LIN {X 0,Y 450.655,Z 566.335,A -85,B 0,C 180,E1 -8884.109,E2 -8884.109} C_VEL
LIN {X 0,Y 449.557,Z 588.314,A -85,B 0,C 180,E1 -8887.411,E2 -8887.411} C_VEL
LIN {X 0,Y 448.704,Z 611.584,A -85,B 0,C 180,E1 -8890.796,E2 -8890.796} C_VEL
LIN {X 0,Y 448.44,Z 622.118,A -85,B 0,C 180,E1 -8892.238,E2 -8892.238} C_VEL
LIN {X 0,Y 450.986,Z 639.711,A -85,B 0,C 180,E1 -8892.631,E2 -8892.631} C_VEL
LIN {X 0,Y 450.667,Z 684.89,A -85,B 0,C 180,E1 -8893.36,E2 -8893.36} C_VEL
LIN {X 0,Y 449.966,Z 688.81,A -85,B 0,C 180,E1 -8893.398,E2 -8893.398} C_VEL
LIN {X 0,Y 444.273,Z 701.08,A -85,B 0,C 180,E1 -8893.381,E2 -8893.381} C_VEL
LIN {X 0,Y 443.65,Z 704.994,A -85,B 0,C 180,E1 -8893.422,E2 -8893.422} C_VEL
LIN {X 0,Y 443.312,Z 733.868,A -85,B 0,C 180,E1 -8893.922,E2 -8893.922} C_VEL
LIN {X 0,Y 442.949,Z 746.723,A -85,B 0,C 180,E1 -8894.322,E2 -8894.322} C_VEL
LIN {X 0,Y 442.385,Z 759.614,A -85,B 0,C 180,E1 -8894.921,E2 -8894.921} C_VEL
LIN {X 0,Y 441.872,Z 770.653,A -85,B 0,C 180,E1 -8895.61,E2 -8895.61} C_VEL
LIN {X 0,Y 441.394,Z 780.851,A -85,B 0,C 180,E1 -8896.417,E2 -8896.417} C_VEL
LIN {X 0,Y 440.796,Z 791.331,A -85,B 0,C 180,E1 -8897.453,E2 -8897.453} C_VEL
LIN {X 0,Y 440.188,Z 799.921,A -85,B 0,C 180,E1 -8898.487,E2 -8898.487} C_VEL
LIN {X 0,Y 439.608,Z 809.259,A -85,B 0,C 180,E1 -8899.871,E2 -8899.871} C_VEL
LIN {X 0,Y 439.155,Z 816.688,A -85,B 0,C 180,E1 -8901.255,E2 -8901.255} C_VEL
LIN {X 0,Y 438.787,Z 822.657,A -85,B 0,C 180,E1 -8902.638,E2 -8902.638} C_VEL
LIN {X 0,Y 438.678,Z 827.373,A -85,B 0,C 180,E1 -8904.022,E2 -8904.022} C_VEL
LIN {X 0,Y 438.409,Z 830.987,A -85,B 0,C 180,E1 -8905.402,E2 -8905.402} C_VEL
LIN {X 0,Y 438.405,Z 832.844,A -85,B 0,C 180,E1 -8906.323,E2 -8906.323} C_VEL
LIN {X 0,Y 438.391,Z 834.266,A -85,B 0,C 180,E1 -8907.243,E2 -8907.243} C_VEL
LIN {X 0,Y 438.255,Z 835.881,A -85,B 0,C 180,E1 -8909.08,E2 -8909.08} C_VEL
LIN {X 0,Y 438.254,Z 836.117,A -85,B 0,C 180,E1 -8909.999,E2 -8909.999} C_VEL
LIN {X 0,Y 438.255,Z 835.929,A -85,B 0,C 180,E1 -8910.918,E2 -8910.918} C_VEL
LIN {X 0,Y 438.391,Z 834.379,A -85,B 0,C 180,E1 -8912.756,E2 -8912.756} C_VEL
LIN {X 0,Y 438.404,Z 833.019,A -85,B 0,C 180,E1 -8913.676,E2 -8913.676} C_VEL
LIN {X 0,Y 438.474,Z 830.154,A -85,B 0,C 180,E1 -8915.057,E2 -8915.057} C_VEL
LIN {X 0,Y 438.686,Z 825.559,A -85,B 0,C 180,E1 -8916.646,E2 -8916.646} C_VEL
LIN {X 0,Y 438.996,Z 819.257,A -85,B 0,C 180,E1 -8918.283,E2 -8918.283} C_VEL
LIN {X 0,Y 439.4,Z 812.443,A -85,B 0,C 180,E1 -8919.667,E2 -8919.667} C_VEL
LIN {X 0,Y 439.914,Z 803.901,A -85,B 0,C 180,E1 -8921.052,E2 -8921.052} C_VEL
LIN {X 0,Y 440.558,Z 795.158,A -85,B 0,C 180,E1 -8922.202,E2 -8922.202} C_VEL
LIN {X 0,Y 441.142,Z 785.519,A -85,B 0,C 180,E1 -8923.243,E2 -8923.243} C_VEL
LIN {X 0,Y 441.716,Z 774.968,A -85,B 0,C 180,E1 -8924.159,E2 -8924.159} C_VEL
LIN {X 0,Y 442.267,Z 763.215,A -85,B 0,C 180,E1 -8924.964,E2 -8924.964} C_VEL
LIN {X 0,Y 442.817,Z 751.05,A -85,B 0,C 180,E1 -8925.593,E2 -8925.593} C_VEL
LIN {X 0,Y 443.202,Z 738.346,A -85,B 0,C 180,E1 -8926.051,E2 -8926.051} C_VEL
LIN {X 0,Y 443.436,Z 725.465,A -85,B 0,C 180,E1 -8926.338,E2 -8926.338} C_VEL
LIN {X 0,Y 444.112,Z 640.098,A -85,B 0,C 180,E1 -8927.734,E2 -8927.734} C_VEL
LIN {X 0,Y 441.171,Z 622.808,A -85,B 0,C 180,E1 -8928.176,E2 -8928.176} C_VEL
LIN {X 0,Y 441.634,Z 608.028,A -85,B 0,C 180,E1 -8930.492,E2 -8930.492} C_VEL
LIN {X 0,Y 442.46,Z 588.945,A -85,B 0,C 180,E1 -8933.644,E2 -8933.644} C_VEL
LIN {X 0,Y 443.197,Z 571.508,A -85,B 0,C 180,E1 -8936.613,E2 -8936.613} C_VEL
LIN {X 0,Y 443.34,Z 564.171,A -85,B 0,C 180,E1 -8937.88,E2 -8937.88} C_VEL
LIN {X 0,Y 440.924,Z 552.234,A -85,B 0,C 180,E1 -8940.079,E2 -8940.079} C_VEL
LIN {X 0,Y 439.385,Z 545.753,A -85,B 0,C 180,E1 -8941.32,E2 -8941.32} C_VEL
LIN {X 0,Y 439.385,Z 545.755,A -85,B 0,C 180,E1 -8944.042,E2 -8944.042} C_VEL
LIN {X 0,Y 439.354,Z 545.757,A -85,B 0,C 180,E1 -8946.888,E2 -8946.888} C_VEL
LIN {X 0,Y 439.409,Z 545.747,A -85,B 0,C 180,E1 -8949.85,E2 -8949.85} C_VEL
LIN {X 0,Y 439.381,Z 545.75,A -85,B 0,C 180,E1 -8952.626,E2 -8952.626} C_VEL
LIN {X 0,Y 439.397,Z 545.75,A -85,B 0,C 180,E1 -8956.032,E2 -8956.032} C_VEL
LIN {X 0,Y 439.394,Z 545.754,A -85,B 0,C 180,E1 -8959.021,E2 -8959.021} C_VEL
LIN {X 0,Y 439.464,Z 545.804,A -85,B 0,C 180,E1 -8960.616,E2 -8960.616} C_VEL
LIN {X 0,Y 443.64,Z 558.186,A -85,B 0,C 180,E1 -8961.004,E2 -8961.004} C_VEL
LIN {X 0,Y 442.996,Z 626.253,A -85,B 0,C 180,E1 -8962.231,E2 -8962.231} C_VEL
LIN {X 0,Y 442.904,Z 640.237,A -85,B 0,C 180,E1 -8962.685,E2 -8962.685} C_VEL
LIN {X 0,Y 442.685,Z 652.211,A -85,B 0,C 180,E1 -8963.25,E2 -8963.25} C_VEL
LIN {X 0,Y 442.358,Z 664.004,A -85,B 0,C 180,E1 -8963.996,E2 -8963.996} C_VEL
LIN {X 0,Y 441.89,Z 675.616,A -85,B 0,C 180,E1 -8964.932,E2 -8964.932} C_VEL
LIN {X 0,Y 441.419,Z 685.917,A -85,B 0,C 180,E1 -8965.971,E2 -8965.971} C_VEL
LIN {X 0,Y 440.931,Z 695.582,A -85,B 0,C 180,E1 -8967.185,E2 -8967.185} C_VEL
LIN {X 0,Y 440.551,Z 704.101,A -85,B 0,C 180,E1 -8968.503,E2 -8968.503} C_VEL
LIN {X 0,Y 440.109,Z 711.544,A -85,B 0,C 180,E1 -8969.937,E2 -8969.937} C_VEL
LIN {X 0,Y 439.77,Z 717.941,A -85,B 0,C 180,E1 -8971.514,E2 -8971.514} C_VEL
LIN {X 0,Y 439.6,Z 722.254,A -85,B 0,C 180,E1 -8972.894,E2 -8972.894} C_VEL
LIN {X 0,Y 439.415,Z 725.795,A -85,B 0,C 180,E1 -8974.416,E2 -8974.416} C_VEL
LIN {X 0,Y 439.289,Z 727.92,A -85,B 0,C 180,E1 -8975.768,E2 -8975.768} C_VEL
LIN {X 0,Y 439.282,Z 729.321,A -85,B 0,C 180,E1 -8977.42,E2 -8977.42} C_VEL
LIN {X 0,Y 439.291,Z 729.501,A -85,B 0,C 180,E1 -8978.41,E2 -8978.41} C_VEL
LIN {X 0,Y 439.353,Z 729.247,A -85,B 0,C 180,E1 -8979.395,E2 -8979.395} C_VEL
LIN {X 0,Y 439.471,Z 728.221,A -85,B 0,C 180,E1 -8980.647,E2 -8980.647} C_VEL
LIN {X 0,Y 439.647,Z 725.684,A -85,B 0,C 180,E1 -8982.318,E2 -8982.318} C_VEL
LIN {X 0,Y 439.923,Z 722.044,A -85,B 0,C 180,E1 -8983.85,E2 -8983.85} C_VEL
LIN {X 0,Y 440.238,Z 717.703,A -85,B 0,C 180,E1 -8985.201,E2 -8985.201} C_VEL
LIN {X 0,Y 440.71,Z 710.974,A -85,B 0,C 180,E1 -8986.807,E2 -8986.807} C_VEL
LIN {X 0,Y 441.129,Z 704.434,A -85,B 0,C 180,E1 -8988.047,E2 -8988.047} C_VEL
LIN {X 0,Y 441.614,Z 696.861,A -85,B 0,C 180,E1 -8989.223,E2 -8989.223} C_VEL
LIN {X 0,Y 442.106,Z 687.903,A -85,B 0,C 180,E1 -8990.362,E2 -8990.362} C_VEL
LIN {X 0,Y 442.623,Z 677.349,A -85,B 0,C 180,E1 -8991.439,E2 -8991.439} C_VEL
LIN {X 0,Y 443.073,Z 665.968,A -85,B 0,C 180,E1 -8992.366,E2 -8992.366} C_VEL
LIN {X 0,Y 443.499,Z 653.859,A -85,B 0,C 180,E1 -8993.117,E2 -8993.117} C_VEL
LIN {X 0,Y 443.659,Z 640.811,A -85,B 0,C 180,E1 -8993.719,E2 -8993.719} C_VEL
LIN {X 0,Y 443.726,Z 628.913,A -85,B 0,C 180,E1 -8994.091,E2 -8994.091} C_VEL
LIN {X 0,Y 444.376,Z 571.276,A -85,B 0,C 180,E1 -8995.165,E2 -8995.165} C_VEL
LIN {X 0,Y 444.368,Z 558.239,A -85,B 0,C 180,E1 -8995.419,E2 -8995.419} C_VEL
LIN {X 0,Y 439.515,Z 546.251,A -85,B 0,C 180,E1 -8995.902,E2 -8995.902} C_VEL
LIN {X 0,Y 439.442,Z 545.747,A -85,B 0,C 180,E1 -8995.93,E2 -8995.93} C_VEL
LIN {X 0,Y 439.627,Z 545.725,A -85,B 0,C 180,E1 -8998.168,E2 -8998.168} C_VEL
LIN {X 0,Y 439.754,Z 545.709,A -85,B 0,C 180,E1 -9000,E2 -9000} C_VEL
LIN {X 0,Y 439.647,Z 545.724,A -85,B 0,C 180,E1 -9002.749,E2 -9002.749} C_VEL
LIN {X 0,Y 439.612,Z 545.726,A -85,B 0,C 180,E1 -9006.425,E2 -9006.425} C_VEL
LIN {X 0,Y 439.491,Z 545.738,A -85,B 0,C 180,E1 -9009.202,E2 -9009.202} C_VEL
LIN {X 0,Y 439.493,Z 545.738,A -85,B 0,C 180,E1 -9012.727,E2 -9012.727} C_VEL
LIN {X 0,Y 439.436,Z 545.742,A -85,B 0,C 180,E1 -9016.349,E2 -9016.349} C_VEL
LIN {X 0,Y 439.392,Z 545.749,A -85,B 0,C 180,E1 -9019.627,E2 -9019.627} C_VEL
LIN {X 0,Y 439.355,Z 545.76,A -85,B 0,C 180,E1 -9022.576,E2 -9022.576} C_VEL
LIN {X 0,Y 439.395,Z 545.749,A -85,B 0,C 180,E1 -9025.586,E2 -9025.586} C_VEL
LIN {X 0,Y 439.416,Z 545.752,A -85,B 0,C 180,E1 -9028.674,E2 -9028.674} C_VEL
LIN {X 0,Y 439.366,Z 545.753,A -85,B 0,C 180,E1 -9031.861,E2 -9031.861} C_VEL
LIN {X 0,Y 439.393,Z 545.752,A -85,B 0,C 180,E1 -9035.157,E2 -9035.157} C_VEL
LIN {X 0,Y 439.392,Z 545.753,A -85,B 0,C 180,E1 -9038.594,E2 -9038.594} C_VEL
LIN {X 0,Y 439.398,Z 545.754,A -85,B 0,C 180,E1 -9041.26,E2 -9041.26} C_VEL
LIN {X 0,Y 439.404,Z 545.753,A -85,B 0,C 180,E1 -9044.729,E2 -9044.729} C_VEL
LIN {X 0,Y 439.407,Z 545.749,A -85,B 0,C 180,E1 -9047.799,E2 -9047.799} C_VEL
LIN {X 0,Y 439.447,Z 545.746,A -85,B 0,C 180,E1 -9050.231,E2 -9050.231} C_VEL
LIN {X 0,Y 439.374,Z 545.757,A -85,B 0,C 180,E1 -9053.714,E2 -9053.714} C_VEL
LIN {X 0,Y 439.369,Z 545.758,A -85,B 0,C 180,E1 -9057.055,E2 -9057.055} C_VEL
LIN {X 0,Y 439.402,Z 545.859,A -85,B 0,C 180,E1 -9058.345,E2 -9058.345} C_VEL
LIN {X 0,Y 442.762,Z 559.87,A -85,B 0,C 180,E1 -9060.812,E2 -9060.812} C_VEL
LIN {X 0,Y 443.906,Z 566.478,A -85,B 0,C 180,E1 -9061.901,E2 -9061.901} C_VEL
LIN {X 0,Y 442.686,Z 586.17,A -85,B 0,C 180,E1 -9064.813,E2 -9064.813} C_VEL
LIN {X 0,Y 441.546,Z 608.576,A -85,B 0,C 180,E1 -9068.036,E2 -9068.036} C_VEL
LIN {X 0,Y 440.516,Z 632.39,A -85,B 0,C 180,E1 -9071.394,E2 -9071.394} C_VEL
LIN {X 0,Y 440.424,Z 634.814,A -85,B 0,C 180,E1 -9071.721,E2 -9071.721} C_VEL
LIN {X 0,Y 443.782,Z 667.711,A -85,B 0,C 180,E1 -9072.49,E2 -9072.49} C_VEL
LIN {X 0,Y 442.669,Z 758.735,A -85,B 0,C 180,E1 -9074.106,E2 -9074.106} C_VEL
LIN {X 0,Y 442.256,Z 772.248,A -85,B 0,C 180,E1 -9074.535,E2 -9074.535} C_VEL
LIN {X 0,Y 441.746,Z 784.913,A -85,B 0,C 180,E1 -9075.136,E2 -9075.136} C_VEL
LIN {X 0,Y 441.183,Z 797.312,A -85,B 0,C 180,E1 -9075.941,E2 -9075.941} C_VEL
LIN {X 0,Y 440.675,Z 807.744,A -85,B 0,C 180,E1 -9076.809,E2 -9076.809} C_VEL
LIN {X 0,Y 440.121,Z 817.257,A -85,B 0,C 180,E1 -9077.786,E2 -9077.786} C_VEL
LIN {X 0,Y 439.552,Z 826.395,A -85,B 0,C 180,E1 -9078.939,E2 -9078.939} C_VEL
LIN {X 0,Y 439.082,Z 835.281,A -85,B 0,C 180,E1 -9080.326,E2 -9080.326} C_VEL
LIN {X 0,Y 438.787,Z 842.39,A -85,B 0,C 180,E1 -9081.713,E2 -9081.713} C_VEL
LIN {X 0,Y 438.589,Z 848.034,A -85,B 0,C 180,E1 -9083.098,E2 -9083.098} C_VEL
LIN {X 0,Y 438.497,Z 852.458,A -85,B 0,C 180,E1 -9084.482,E2 -9084.482} C_VEL
LIN {X 0,Y 438.432,Z 854.786,A -85,B 0,C 180,E1 -9085.404,E2 -9085.404} C_VEL
LIN {X 0,Y 438.399,Z 856.683,A -85,B 0,C 180,E1 -9086.324,E2 -9086.324} C_VEL
LIN {X 0,Y 438.44,Z 858.116,A -85,B 0,C 180,E1 -9087.244,E2 -9087.244} C_VEL
LIN {X 0,Y 438.384,Z 859.74,A -85,B 0,C 180,E1 -9089.082,E2 -9089.082} C_VEL
LIN {X 0,Y 438.403,Z 859.961,A -85,B 0,C 180,E1 -9090.001,E2 -9090.001} C_VEL
LIN {X 0,Y 438.368,Z 859.12,A -85,B 0,C 180,E1 -9091.838,E2 -9091.838} C_VEL
LIN {X 0,Y 438.428,Z 858.111,A -85,B 0,C 180,E1 -9092.757,E2 -9092.757} C_VEL
LIN {X 0,Y 438.38,Z 856.675,A -85,B 0,C 180,E1 -9093.677,E2 -9093.677} C_VEL
LIN {X 0,Y 438.479,Z 853.693,A -85,B 0,C 180,E1 -9095.058,E2 -9095.058} C_VEL
LIN {X 0,Y 438.546,Z 849.478,A -85,B 0,C 180,E1 -9096.488,E2 -9096.488} C_VEL
LIN {X 0,Y 438.73,Z 843.383,A -85,B 0,C 180,E1 -9098.058,E2 -9098.058} C_VEL
LIN {X 0,Y 439.04,Z 836.554,A -85,B 0,C 180,E1 -9099.444,E2 -9099.444} C_VEL
LIN {X 0,Y 439.346,Z 829.572,A -85,B 0,C 180,E1 -9100.601,E2 -9100.601} C_VEL
LIN {X 0,Y 439.86,Z 821.133,A -85,B 0,C 180,E1 -9101.755,E2 -9101.755} C_VEL
LIN {X 0,Y 440.44,Z 810.661,A -85,B 0,C 180,E1 -9102.909,E2 -9102.909} C_VEL
LIN {X 0,Y 440.974,Z 800.271,A -85,B 0,C 180,E1 -9103.832,E2 -9103.832} C_VEL
LIN {X 0,Y 441.557,Z 788.805,A -85,B 0,C 180,E1 -9104.636,E2 -9104.636} C_VEL
LIN {X 0,Y 442.081,Z 776.867,A -85,B 0,C 180,E1 -9105.267,E2 -9105.267} C_VEL
LIN {X 0,Y 442.539,Z 763.915,A -85,B 0,C 180,E1 -9105.752,E2 -9105.752} C_VEL
LIN {X 0,Y 442.736,Z 751.562,A -85,B 0,C 180,E1 -9106.04,E2 -9106.04} C_VEL
LIN {X 0,Y 443.494,Z 683.953,A -85,B 0,C 180,E1 -9107.17,E2 -9107.17} C_VEL
LIN {X 0,Y 443.456,Z 667.459,A -85,B 0,C 180,E1 -9107.471,E2 -9107.471} C_VEL
LIN {X 0,Y 440.217,Z 639.525,A -85,B 0,C 180,E1 -9108.107,E2 -9108.107} C_VEL
LIN {X 0,Y 441.018,Z 620.987,A -85,B 0,C 180,E1 -9111.012,E2 -9111.012} C_VEL
LIN {X 0,Y 441.922,Z 602.556,A -85,B 0,C 180,E1 -9113.925,E2 -9113.925} C_VEL
LIN {X 0,Y 443.154,Z 580.99,A -85,B 0,C 180,E1 -9117.382,E2 -9117.382} C_VEL
LIN {X 0,Y 443.949,Z 567.072,A -85,B 0,C 180,E1 -9119.65,E2 -9119.65} C_VEL
LIN {X 0,Y 441.963,Z 556.965,A -85,B 0,C 180,E1 -9121.451,E2 -9121.451} C_VEL
LIN {X 0,Y 439.414,Z 545.751,A -85,B 0,C 180,E1 -9123.55,E2 -9123.55} C_VEL
LIN {X 0,Y 439.376,Z 545.754,A -85,B 0,C 180,E1 -9126.287,E2 -9126.287} C_VEL
LIN {X 0,Y 439.408,Z 545.748,A -85,B 0,C 180,E1 -9129.85,E2 -9129.85} C_VEL
LIN {X 0,Y 439.384,Z 545.753,A -85,B 0,C 180,E1 -9132.627,E2 -9132.627} C_VEL
LIN {X 0,Y 439.408,Z 545.752,A -85,B 0,C 180,E1 -9135.271,E2 -9135.271} C_VEL
LIN {X 0,Y 439.391,Z 545.745,A -85,B 0,C 180,E1 -9138.743,E2 -9138.743} C_VEL
LIN {X 0,Y 439.384,Z 545.75,A -85,B 0,C 180,E1 -9141.606,E2 -9141.606} C_VEL
LIN {X 0,Y 439.402,Z 545.746,A -85,B 0,C 180,E1 -9144.844,E2 -9144.844} C_VEL
LIN {X 0,Y 439.373,Z 545.745,A -85,B 0,C 180,E1 -9148.139,E2 -9148.139} C_VEL
LIN {X 0,Y 439.433,Z 545.748,A -85,B 0,C 180,E1 -9151.598,E2 -9151.598} C_VEL
LIN {X 0,Y 439.405,Z 545.74,A -85,B 0,C 180,E1 -9154.415,E2 -9154.415} C_VEL
LIN {X 0,Y 439.365,Z 545.755,A -85,B 0,C 180,E1 -9157.425,E2 -9157.425} C_VEL
LIN {X 0,Y 439.442,Z 545.739,A -85,B 0,C 180,E1 -9160.663,E2 -9160.663} C_VEL
LIN {X 0,Y 439.463,Z 545.738,A -85,B 0,C 180,E1 -9164.225,E2 -9164.225} C_VEL
LIN {X 0,Y 439.483,Z 545.731,A -85,B 0,C 180,E1 -9168.001,E2 -9168.001} C_VEL
LIN {X 0,Y 439.548,Z 545.731,A -85,B 0,C 180,E1 -9171.726,E2 -9171.726} C_VEL
LIN {X 0,Y 439.621,Z 545.719,A -85,B 0,C 180,E1 -9174.496,E2 -9174.496} C_VEL
LIN {X 0,Y 439.634,Z 545.714,A -85,B 0,C 180,E1 -9178.168,E2 -9178.168} C_VEL
LIN {X 0,Y 439.762,Z 545.706,A -85,B 0,C 180,E1 -9180,E2 -9180} C_VEL
LIN {X 0,Y 439.641,Z 545.715,A -85,B 0,C 180,E1 -9182.749,E2 -9182.749} C_VEL
LIN {X 0,Y 439.618,Z 545.717,A -85,B 0,C 180,E1 -9186.425,E2 -9186.425} C_VEL
LIN {X 0,Y 439.5,Z 545.737,A -85,B 0,C 180,E1 -9189.202,E2 -9189.202} C_VEL
LIN {X 0,Y 439.466,Z 545.728,A -85,B 0,C 180,E1 -9192.938,E2 -9192.938} C_VEL
LIN {X 0,Y 439.448,Z 545.743,A -85,B 0,C 180,E1 -9196.349,E2 -9196.349} C_VEL
LIN {X 0,Y 439.403,Z 545.74,A -85,B 0,C 180,E1 -9199.626,E2 -9199.626} C_VEL
LIN {X 0,Y 439.366,Z 545.753,A -85,B 0,C 180,E1 -9202.576,E2 -9202.576} C_VEL
LIN {X 0,Y 439.406,Z 545.741,A -85,B 0,C 180,E1 -9205.585,E2 -9205.585} C_VEL
LIN {X 0,Y 439.418,Z 545.746,A -85,B 0,C 180,E1 -9208.674,E2 -9208.674} C_VEL
LIN {X 0,Y 439.371,Z 545.753,A -85,B 0,C 180,E1 -9212.03,E2 -9212.03} C_VEL
LIN {X 0,Y 439.395,Z 545.745,A -85,B 0,C 180,E1 -9215.34,E2 -9215.34} C_VEL
LIN {X 0,Y 439.38,Z 545.752,A -85,B 0,C 180,E1 -9218.596,E2 -9218.596} C_VEL
LIN {X 0,Y 439.39,Z 545.751,A -85,B 0,C 180,E1 -9221.257,E2 -9221.257} C_VEL
LIN {X 0,Y 439.401,Z 545.75,A -85,B 0,C 180,E1 -9224.73,E2 -9224.73} C_VEL
LIN {X 0,Y 439.387,Z 545.738,A -85,B 0,C 180,E1 -9227.794,E2 -9227.794} C_VEL
LIN {X 0,Y 439.439,Z 545.75,A -85,B 0,C 180,E1 -9230.228,E2 -9230.228} C_VEL
LIN {X 0,Y 439.377,Z 545.753,A -85,B 0,C 180,E1 -9233.713,E2 -9233.713} C_VEL
LIN {X 0,Y 439.376,Z 545.755,A -85,B 0,C 180,E1 -9237.054,E2 -9237.054} C_VEL
LIN {X 0,Y 439.42,Z 545.891,A -85,B 0,C 180,E1 -9240.343,E2 -9240.343} C_VEL
LIN {X 0,Y 442.753,Z 560.22,A -85,B 0,C 180,E1 -9242.737,E2 -9242.737} C_VEL
LIN {X 0,Y 443.809,Z 565.987,A -85,B 0,C 180,E1 -9243.679,E2 -9243.679} C_VEL
LIN {X 0,Y 442.972,Z 583.794,A -85,B 0,C 180,E1 -9246.384,E2 -9246.384} C_VEL
LIN {X 0,Y 441.928,Z 609.149,A -85,B 0,C 180,E1 -9250.139,E2 -9250.139} C_VEL
LIN {X 0,Y 441.535,Z 622.105,A -85,B 0,C 180,E1 -9251.943,E2 -9251.943} C_VEL
LIN {X 0,Y 444.191,Z 639.141,A -85,B 0,C 180,E1 -9252.346,E2 -9252.346} C_VEL
LIN {X 0,Y 443.65,Z 704.994,A -85,B 0,C 180,E1 -9253.422,E2 -9253.422} C_VEL
LIN {X 0,Y 443.079,Z 710.844,A -85,B 0,C 180,E1 -9253.491,E2 -9253.491} C_VEL
LIN {X 0,Y 437.308,Z 729.831,A -85,B 0,C 180,E1 -9253.589,E2 -9253.589} C_VEL
LIN {X 0,Y 436.482,Z 735.621,A -85,B 0,C 180,E1 -9253.704,E2 -9253.704} C_VEL
LIN {X 0,Y 436.044,Z 748.989,A -85,B 0,C 180,E1 -9254.157,E2 -9254.157} C_VEL
LIN {X 0,Y 435.508,Z 760.848,A -85,B 0,C 180,E1 -9254.737,E2 -9254.737} C_VEL
LIN {X 0,Y 434.919,Z 772.429,A -85,B 0,C 180,E1 -9255.494,E2 -9255.494} C_VEL
LIN {X 0,Y 434.387,Z 783.2,A -85,B 0,C 180,E1 -9256.4,E2 -9256.4} C_VEL
LIN {X 0,Y 433.73,Z 793.584,A -85,B 0,C 180,E1 -9257.483,E2 -9257.483} C_VEL
LIN {X 0,Y 433.145,Z 801.836,A -85,B 0,C 180,E1 -9258.535,E2 -9258.535} C_VEL
LIN {X 0,Y 432.53,Z 810.78,A -85,B 0,C 180,E1 -9259.94,E2 -9259.94} C_VEL
LIN {X 0,Y 432.048,Z 817.968,A -85,B 0,C 180,E1 -9261.345,E2 -9261.345} C_VEL
LIN {X 0,Y 431.674,Z 824.57,A -85,B 0,C 180,E1 -9262.986,E2 -9262.986} C_VEL
LIN {X 0,Y 431.527,Z 828.898,A -85,B 0,C 180,E1 -9264.392,E2 -9264.392} C_VEL
LIN {X 0,Y 431.339,Z 831.18,A -85,B 0,C 180,E1 -9265.326,E2 -9265.326} C_VEL
LIN {X 0,Y 431.31,Z 833.038,A -85,B 0,C 180,E1 -9266.262,E2 -9266.262} C_VEL
LIN {X 0,Y 431.322,Z 834.459,A -85,B 0,C 180,E1 -9267.197,E2 -9267.197} C_VEL
LIN {X 0,Y 431.172,Z 836.074,A -85,B 0,C 180,E1 -9269.065,E2 -9269.065} C_VEL
LIN {X 0,Y 431.168,Z 836.31,A -85,B 0,C 180,E1 -9269.999,E2 -9269.999} C_VEL
LIN {X 0,Y 431.172,Z 836.121,A -85,B 0,C 180,E1 -9270.933,E2 -9270.933} C_VEL
LIN {X 0,Y 431.322,Z 834.57,A -85,B 0,C 180,E1 -9272.801,E2 -9272.801} C_VEL
LIN {X 0,Y 431.309,Z 833.211,A -85,B 0,C 180,E1 -9273.736,E2 -9273.736} C_VEL
LIN {X 0,Y 431.42,Z 830.345,A -85,B 0,C 180,E1 -9275.14,E2 -9275.14} C_VEL
LIN {X 0,Y 431.613,Z 826.102,A -85,B 0,C 180,E1 -9276.649,E2 -9276.649} C_VEL
LIN {X 0,Y 431.859,Z 821.409,A -85,B 0,C 180,E1 -9277.95,E2 -9277.95} C_VEL
LIN {X 0,Y 432.263,Z 815.052,A -85,B 0,C 180,E1 -9279.356,E2 -9279.356} C_VEL
LIN {X 0,Y 432.79,Z 807.143,A -85,B 0,C 180,E1 -9280.762,E2 -9280.762} C_VEL
LIN {X 0,Y 433.298,Z 799.06,A -85,B 0,C 180,E1 -9281.934,E2 -9281.934} C_VEL
LIN {X 0,Y 434.05,Z 789.143,A -85,B 0,C 180,E1 -9283.101,E2 -9283.101} C_VEL
LIN {X 0,Y 434.641,Z 778.007,A -85,B 0,C 180,E1 -9284.155,E2 -9284.155} C_VEL
LIN {X 0,Y 435.253,Z 767.102,A -85,B 0,C 180,E1 -9284.971,E2 -9284.971} C_VEL
LIN {X 0,Y 435.767,Z 756.077,A -85,B 0,C 180,E1 -9285.612,E2 -9285.612} C_VEL
LIN {X 0,Y 436.259,Z 743.003,A -85,B 0,C 180,E1 -9286.163,E2 -9286.163} C_VEL
LIN {X 0,Y 436.533,Z 730.329,A -85,B 0,C 180,E1 -9286.513,E2 -9286.513} C_VEL
LIN {X 0,Y 437.423,Z 641.442,A -85,B 0,C 180,E1 -9287.992,E2 -9287.992} C_VEL
LIN {X 0,Y 434.295,Z 623.142,A -85,B 0,C 180,E1 -9288.442,E2 -9288.442} C_VEL
LIN {X 0,Y 434.744,Z 609.057,A -85,B 0,C 180,E1 -9290.658,E2 -9290.658} C_VEL
LIN {X 0,Y 435.559,Z 590.228,A -85,B 0,C 180,E1 -9293.789,E2 -9293.789} C_VEL
LIN {X 0,Y 436.445,Z 571.304,A -85,B 0,C 180,E1 -9297.038,E2 -9297.038} C_VEL
LIN {X 0,Y 436.558,Z 566.734,A -85,B 0,C 180,E1 -9297.829,E2 -9297.829} C_VEL
LIN {X 0,Y 434.785,Z 557.146,A -85,B 0,C 180,E1 -9299.608,E2 -9299.608} C_VEL
LIN {X 0,Y 432.344,Z 546.629,A -85,B 0,C 180,E1 -9301.616,E2 -9301.616} C_VEL
LIN {X 0,Y 432.338,Z 546.634,A -85,B 0,C 180,E1 -9304.676,E2 -9304.676} C_VEL
LIN {X 0,Y 432.344,Z 546.632,A -85,B 0,C 180,E1 -9308.148,E2 -9308.148} C_VEL
LIN {X 0,Y 432.329,Z 546.632,A -85,B 0,C 180,E1 -9311.601,E2 -9311.601} C_VEL
LIN {X 0,Y 432.336,Z 546.622,A -85,B 0,C 180,E1 -9314.345,E2 -9314.345} C_VEL
LIN {X 0,Y 432.36,Z 546.629,A -85,B 0,C 180,E1 -9317.008,E2 -9317.008} C_VEL
LIN {X 0,Y 432.41,Z 546.622,A -85,B 0,C 180,E1 -9320.344,E2 -9320.344} C_VEL
LIN {X 0,Y 436.956,Z 560.3,A -85,B 0,C 180,E1 -9320.793,E2 -9320.793} C_VEL
LIN {X 0,Y 436.114,Z 627.319,A -85,B 0,C 180,E1 -9322.019,E2 -9322.019} C_VEL
LIN {X 0,Y 436.048,Z 641.37,A -85,B 0,C 180,E1 -9322.487,E2 -9322.487} C_VEL
LIN {X 0,Y 435.813,Z 653.599,A -85,B 0,C 180,E1 -9323.08,E2 -9323.08} C_VEL
LIN {X 0,Y 435.405,Z 666.168,A -85,B 0,C 180,E1 -9323.9,E2 -9323.9} C_VEL
LIN {X 0,Y 434.927,Z 677.59,A -85,B 0,C 180,E1 -9324.854,E2 -9324.854} C_VEL
LIN {X 0,Y 434.445,Z 687.92,A -85,B 0,C 180,E1 -9325.941,E2 -9325.941} C_VEL
LIN {X 0,Y 433.907,Z 698.229,A -85,B 0,C 180,E1 -9327.287,E2 -9327.287} C_VEL
LIN {X 0,Y 433.541,Z 705.62,A -85,B 0,C 180,E1 -9328.48,E2 -9328.48} C_VEL
LIN {X 0,Y 433.127,Z 712.34,A -85,B 0,C 180,E1 -9329.8,E2 -9329.8} C_VEL
LIN {X 0,Y 432.786,Z 718.311,A -85,B 0,C 180,E1 -9331.268,E2 -9331.268} C_VEL
LIN {X 0,Y 432.593,Z 723.521,A -85,B 0,C 180,E1 -9332.942,E2 -9332.942} C_VEL
LIN {X 0,Y 432.432,Z 725.955,A -85,B 0,C 180,E1 -9333.972,E2 -9333.972} C_VEL
LIN {X 0,Y 432.286,Z 728.668,A -85,B 0,C 180,E1 -9335.561,E2 -9335.561} C_VEL
LIN {X 0,Y 432.257,Z 730.101,A -85,B 0,C 180,E1 -9337.032,E2 -9337.032} C_VEL
LIN {X 0,Y 432.297,Z 730.517,A -85,B 0,C 180,E1 -9338.042,E2 -9338.042} C_VEL
LIN {X 0,Y 432.311,Z 730.435,A -85,B 0,C 180,E1 -9339.044,E2 -9339.044} C_VEL
LIN {X 0,Y 432.441,Z 729.503,A -85,B 0,C 180,E1 -9340.49,E2 -9340.49} C_VEL
LIN {X 0,Y 432.609,Z 727.429,A -85,B 0,C 180,E1 -9342.021,E2 -9342.021} C_VEL
LIN {X 0,Y 432.858,Z 724.765,A -85,B 0,C 180,E1 -9343.318,E2 -9343.318} C_VEL
LIN {X 0,Y 433.213,Z 720.074,A -85,B 0,C 180,E1 -9344.956,E2 -9344.956} C_VEL
LIN {X 0,Y 433.686,Z 714.268,A -85,B 0,C 180,E1 -9346.48,E2 -9346.48} C_VEL
LIN {X 0,Y 434.107,Z 707.636,A -85,B 0,C 180,E1 -9347.85,E2 -9347.85} C_VEL
LIN {X 0,Y 434.718,Z 698.857,A -85,B 0,C 180,E1 -9349.285,E2 -9349.285} C_VEL
LIN {X 0,Y 435.217,Z 690.387,A -85,B 0,C 180,E1 -9350.408,E2 -9350.408} C_VEL
LIN {X 0,Y 435.757,Z 679.864,A -85,B 0,C 180,E1 -9351.537,E2 -9351.537} C_VEL
LIN {X 0,Y 436.255,Z 668.768,A -85,B 0,C 180,E1 -9352.479,E2 -9352.479} C_VEL
LIN {X 0,Y 436.645,Z 658.272,A -85,B 0,C 180,E1 -9353.183,E2 -9353.183} C_VEL
LIN {X 0,Y 436.898,Z 645.833,A -85,B 0,C 180,E1 -9353.824,E2 -9353.824} C_VEL
LIN {X 0,Y 436.972,Z 632.79,A -85,B 0,C 180,E1 -9354.289,E2 -9354.289} C_VEL
LIN {X 0,Y 437.024,Z 612.359,A -85,B 0,C 180,E1 -9354.717,E2 -9354.717} C_VEL
LIN {X 0,Y 437.812,Z 560.181,A -85,B 0,C 180,E1 -9355.707,E2 -9355.707} C_VEL
LIN {X 0,Y 432.492,Z 547.212,A -85,B 0,C 180,E1 -9356.249,E2 -9356.249} C_VEL
LIN {X 0,Y 432.404,Z 546.626,A -85,B 0,C 180,E1 -9356.272,E2 -9356.272} C_VEL
LIN {X 0,Y 432.597,Z 546.601,A -85,B 0,C 180,E1 -9358.138,E2 -9358.138} C_VEL
LIN {X 0,Y 432.724,Z 546.585,A -85,B 0,C 180,E1 -9360,E2 -9360} C_VEL
LIN {X 0,Y 432.597,Z 546.602,A -85,B 0,C 180,E1 -9362.794,E2 -9362.794} C_VEL
LIN {X 0,Y 432.566,Z 546.606,A -85,B 0,C 180,E1 -9366.53,E2 -9366.53} C_VEL
LIN {X 0,Y 432.434,Z 546.616,A -85,B 0,C 180,E1 -9369.353,E2 -9369.353} C_VEL
LIN {X 0,Y 432.434,Z 546.617,A -85,B 0,C 180,E1 -9372.812,E2 -9372.812} C_VEL
LIN {X 0,Y 432.402,Z 546.62,A -85,B 0,C 180,E1 -9376.479,E2 -9376.479} C_VEL
LIN {X 0,Y 432.329,Z 546.629,A -85,B 0,C 180,E1 -9379.961,E2 -9379.961} C_VEL
LIN {X 0,Y 432.309,Z 546.636,A -85,B 0,C 180,E1 -9382.965,E2 -9382.965} C_VEL
LIN {X 0,Y 432.355,Z 546.626,A -85,B 0,C 180,E1 -9386.033,E2 -9386.033} C_VEL
LIN {X 0,Y 432.343,Z 546.631,A -85,B 0,C 180,E1 -9389.188,E2 -9389.188} C_VEL
LIN {X 0,Y 432.317,Z 546.633,A -85,B 0,C 180,E1 -9392.294,E2 -9392.294} C_VEL
LIN {X 0,Y 432.333,Z 546.629,A -85,B 0,C 180,E1 -9394.678,E2 -9394.678} C_VEL
LIN {X 0,Y 432.346,Z 546.626,A -85,B 0,C 180,E1 -9398.149,E2 -9398.149} C_VEL
LIN {X 0,Y 432.366,Z 546.627,A -85,B 0,C 180,E1 -9401.609,E2 -9401.609} C_VEL
LIN {X 0,Y 432.372,Z 546.629,A -85,B 0,C 180,E1 -9404.343,E2 -9404.343} C_VEL
LIN {X 0,Y 432.36,Z 546.629,A -85,B 0,C 180,E1 -9407.01,E2 -9407.01} C_VEL
LIN {X 0,Y 432.354,Z 546.628,A -85,B 0,C 180,E1 -9409.818,E2 -9409.818} C_VEL
LIN {X 0,Y 432.314,Z 546.639,A -85,B 0,C 180,E1 -9413.024,E2 -9413.024} C_VEL
LIN {X 0,Y 432.356,Z 546.63,A -85,B 0,C 180,E1 -9415.998,E2 -9415.998} C_VEL
LIN {X 0,Y 432.34,Z 546.756,A -85,B 0,C 180,E1 -9417.985,E2 -9417.985} C_VEL
LIN {X 0,Y 435.562,Z 559.807,A -85,B 0,C 180,E1 -9420.358,E2 -9420.358} C_VEL
LIN {X 0,Y 437.024,Z 567.545,A -85,B 0,C 180,E1 -9421.681,E2 -9421.681} C_VEL
LIN {X 0,Y 435.892,Z 585.859,A -85,B 0,C 180,E1 -9424.45,E2 -9424.45} C_VEL
LIN {X 0,Y 434.574,Z 609.446,A -85,B 0,C 180,E1 -9427.915,E2 -9427.915} C_VEL
LIN {X 0,Y 433.465,Z 633.432,A -85,B 0,C 180,E1 -9431.366,E2 -9431.366} C_VEL
LIN {X 0,Y 436.199,Z 659.316,A -85,B 0,C 180,E1 -9432.006,E2 -9432.006} C_VEL
LIN {X 0,Y 437.03,Z 669.777,A -85,B 0,C 180,E1 -9432.243,E2 -9432.243} C_VEL
LIN {X 0,Y 435.839,Z 758.632,A -85,B 0,C 180,E1 -9433.851,E2 -9433.851} C_VEL
LIN {X 0,Y 435.418,Z 772.109,A -85,B 0,C 180,E1 -9434.285,E2 -9434.285} C_VEL
LIN {X 0,Y 434.871,Z 784.752,A -85,B 0,C 180,E1 -9434.896,E2 -9434.896} C_VEL
LIN {X 0,Y 434.281,Z 797.142,A -85,B 0,C 180,E1 -9435.713,E2 -9435.713} C_VEL
LIN {X 0,Y 433.693,Z 808.441,A -85,B 0,C 180,E1 -9436.677,E2 -9436.677} C_VEL
LIN {X 0,Y 433.168,Z 817.076,A -85,B 0,C 180,E1 -9437.587,E2 -9437.587} C_VEL
LIN {X 0,Y 432.571,Z 826.21,A -85,B 0,C 180,E1 -9438.758,E2 -9438.758} C_VEL
LIN {X 0,Y 432.06,Z 835.094,A -85,B 0,C 180,E1 -9440.167,E2 -9440.167} C_VEL
LIN {X 0,Y 431.722,Z 842.2,A -85,B 0,C 180,E1 -9441.576,E2 -9441.576} C_VEL
LIN {X 0,Y 431.52,Z 847.843,A -85,B 0,C 180,E1 -9442.985,E2 -9442.985} C_VEL
LIN {X 0,Y 431.391,Z 852.266,A -85,B 0,C 180,E1 -9444.391,E2 -9444.391} C_VEL
LIN {X 0,Y 431.359,Z 854.595,A -85,B 0,C 180,E1 -9445.328,E2 -9445.328} C_VEL
LIN {X 0,Y 431.299,Z 856.49,A -85,B 0,C 180,E1 -9446.264,E2 -9446.264} C_VEL
LIN {X 0,Y 431.347,Z 857.923,A -85,B 0,C 180,E1 -9447.199,E2 -9447.199} C_VEL
LIN {X 0,Y 431.294,Z 859.547,A -85,B 0,C 180,E1 -9449.067,E2 -9449.067} C_VEL
LIN {X 0,Y 431.309,Z 859.768,A -85,B 0,C 180,E1 -9450.001,E2 -9450.001} C_VEL
LIN {X 0,Y 431.288,Z 858.927,A -85,B 0,C 180,E1 -9451.868,E2 -9451.868} C_VEL
LIN {X 0,Y 431.336,Z 857.918,A -85,B 0,C 180,E1 -9452.803,E2 -9452.803} C_VEL
LIN {X 0,Y 431.282,Z 856.482,A -85,B 0,C 180,E1 -9453.738,E2 -9453.738} C_VEL
LIN {X 0,Y 431.388,Z 853.5,A -85,B 0,C 180,E1 -9455.142,E2 -9455.142} C_VEL
LIN {X 0,Y 431.466,Z 849.448,A -85,B 0,C 180,E1 -9456.548,E2 -9456.548} C_VEL
LIN {X 0,Y 431.684,Z 843.191,A -85,B 0,C 180,E1 -9458.191,E2 -9458.191} C_VEL
LIN {X 0,Y 431.993,Z 836.363,A -85,B 0,C 180,E1 -9459.6,E2 -9459.6} C_VEL
LIN {X 0,Y 432.346,Z 829.383,A -85,B 0,C 180,E1 -9460.775,E2 -9460.775} C_VEL
LIN {X 0,Y 432.875,Z 820.945,A -85,B 0,C 180,E1 -9461.947,E2 -9461.947} C_VEL
LIN {X 0,Y 433.5,Z 810.478,A -85,B 0,C 180,E1 -9463.119,E2 -9463.119} C_VEL
LIN {X 0,Y 434.061,Z 800.091,A -85,B 0,C 180,E1 -9464.057,E2 -9464.057} C_VEL
LIN {X 0,Y 434.666,Z 788.633,A -85,B 0,C 180,E1 -9464.874,E2 -9464.874} C_VEL
LIN {X 0,Y 435.246,Z 776.706,A -85,B 0,C 180,E1 -9465.512,E2 -9465.512} C_VEL
LIN {X 0,Y 435.696,Z 763.774,A -85,B 0,C 180,E1 -9466.006,E2 -9466.006} C_VEL
LIN {X 0,Y 435.918,Z 751.483,A -85,B 0,C 180,E1 -9466.298,E2 -9466.298} C_VEL
LIN {X 0,Y 436.767,Z 669.704,A -85,B 0,C 180,E1 -9467.667,E2 -9467.667} C_VEL
LIN {X 0,Y 433.246,Z 638.609,A -85,B 0,C 180,E1 -9468.392,E2 -9468.392} C_VEL
LIN {X 0,Y 434.144,Z 618.42,A -85,B 0,C 180,E1 -9471.61,E2 -9471.61} C_VEL
LIN {X 0,Y 435.309,Z 596.998,A -85,B 0,C 180,E1 -9475.071,E2 -9475.071} C_VEL
LIN {X 0,Y 436.633,Z 575.382,A -85,B 0,C 180,E1 -9478.611,E2 -9478.611} C_VEL
LIN {X 0,Y 436.918,Z 567.595,A -85,B 0,C 180,E1 -9479.911,E2 -9479.911} C_VEL
LIN {X 0,Y 434.564,Z 556.282,A -85,B 0,C 180,E1 -9481.982,E2 -9481.982} C_VEL
LIN {X 0,Y 432.372,Z 546.627,A -85,B 0,C 180,E1 -9483.841,E2 -9483.841} C_VEL
LIN {X 0,Y 432.325,Z 546.636,A -85,B 0,C 180,E1 -9487.197,E2 -9487.197} C_VEL
LIN {X 0,Y 432.338,Z 546.629,A -85,B 0,C 180,E1 -9490.18,E2 -9490.18} C_VEL
LIN {X 0,Y 432.319,Z 546.632,A -85,B 0,C 180,E1 -9493.061,E2 -9493.061} C_VEL
LIN {X 0,Y 432.344,Z 546.629,A -85,B 0,C 180,E1 -9495.663,E2 -9495.663} C_VEL
LIN {X 0,Y 432.336,Z 546.622,A -85,B 0,C 180,E1 -9498.398,E2 -9498.398} C_VEL
LIN {X 0,Y 432.346,Z 546.625,A -85,B 0,C 180,E1 -9501.851,E2 -9501.851} C_VEL
LIN {X 0,Y 432.342,Z 546.632,A -85,B 0,C 180,E1 -9505.323,E2 -9505.323} C_VEL
LIN {X 0,Y 432.322,Z 546.624,A -85,B 0,C 180,E1 -9508.654,E2 -9508.654} C_VEL
LIN {X 0,Y 432.382,Z 546.624,A -85,B 0,C 180,E1 -9511.877,E2 -9511.877} C_VEL
LIN {X 0,Y 432.352,Z 546.62,A -85,B 0,C 180,E1 -9514.999,E2 -9514.999} C_VEL
LIN {X 0,Y 432.358,Z 546.626,A -85,B 0,C 180,E1 -9518.046,E2 -9518.046} C_VEL
LIN {X 0,Y 432.386,Z 546.62,A -85,B 0,C 180,E1 -9521.03,E2 -9521.03} C_VEL
LIN {X 0,Y 432.431,Z 546.616,A -85,B 0,C 180,E1 -9523.961,E2 -9523.961} C_VEL
LIN {X 0,Y 432.459,Z 546.608,A -85,B 0,C 180,E1 -9527.803,E2 -9527.803} C_VEL
LIN {X 0,Y 432.492,Z 546.607,A -85,B 0,C 180,E1 -9531.59,E2 -9531.59} C_VEL
LIN {X 0,Y 432.598,Z 546.594,A -85,B 0,C 180,E1 -9534.406,E2 -9534.406} C_VEL
LIN {X 0,Y 432.603,Z 546.589,A -85,B 0,C 180,E1 -9538.138,E2 -9538.138} C_VEL
LIN {X 0,Y 432.731,Z 546.582,A -85,B 0,C 180,E1 -9540,E2 -9540} C_VEL
LIN {X 0,Y 432.593,Z 546.593,A -85,B 0,C 180,E1 -9542.794,E2 -9542.794} C_VEL
LIN {X 0,Y 432.573,Z 546.594,A -85,B 0,C 180,E1 -9546.53,E2 -9546.53} C_VEL
LIN {X 0,Y 432.443,Z 546.617,A -85,B 0,C 180,E1 -9549.353,E2 -9549.353} C_VEL
LIN {X 0,Y 432.431,Z 546.604,A -85,B 0,C 180,E1 -9552.803,E2 -9552.803} C_VEL
LIN {X 0,Y 432.413,Z 546.619,A -85,B 0,C 180,E1 -9556.479,E2 -9556.479} C_VEL
LIN {X 0,Y 432.339,Z 546.622,A -85,B 0,C 180,E1 -9559.961,E2 -9559.961} C_VEL
LIN {X 0,Y 432.32,Z 546.63,A -85,B 0,C 180,E1 -9562.964,E2 -9562.964} C_VEL
LIN {X 0,Y 432.365,Z 546.621,A -85,B 0,C 180,E1 -9566.033,E2 -9566.033} C_VEL
LIN {X 0,Y 432.344,Z 546.626,A -85,B 0,C 180,E1 -9569.188,E2 -9569.188} C_VEL
LIN {X 0,Y 432.324,Z 546.635,A -85,B 0,C 180,E1 -9572.443,E2 -9572.443} C_VEL
LIN {X 0,Y 432.345,Z 546.625,A -85,B 0,C 180,E1 -9575.632,E2 -9575.632} C_VEL
LIN {X 0,Y 432.348,Z 546.625,A -85,B 0,C 180,E1 -9579.343,E2 -9579.343} C_VEL
LIN {X 0,Y 432.335,Z 546.633,A -85,B 0,C 180,E1 -9581.797,E2 -9581.797} C_VEL
LIN {X 0,Y 432.335,Z 546.634,A -85,B 0,C 180,E1 -9584.347,E2 -9584.347} C_VEL
LIN {X 0,Y 432.318,Z 546.618,A -85,B 0,C 180,E1 -9587.016,E2 -9587.016} C_VEL
LIN {X 0,Y 432.357,Z 546.626,A -85,B 0,C 180,E1 -9590.658,E2 -9590.658} C_VEL
LIN {X 0,Y 432.348,Z 546.632,A -85,B 0,C 180,E1 -9594.368,E2 -9594.368} C_VEL
LIN {X 0,Y 432.326,Z 546.633,A -85,B 0,C 180,E1 -9597.557,E2 -9597.557} C_VEL
LIN {X 0,Y 432.386,Z 546.819,A -85,B 0,C 180,E1 -9600.046,E2 -9600.046} C_VEL
LIN {X 0,Y 435.79,Z 561.32,A -85,B 0,C 180,E1 -9602.498,E2 -9602.498} C_VEL
LIN {X 0,Y 436.958,Z 567.279,A -85,B 0,C 180,E1 -9603.491,E2 -9603.491} C_VEL
LIN {X 0,Y 436.206,Z 583.598,A -85,B 0,C 180,E1 -9605.994,E2 -9605.994} C_VEL
LIN {X 0,Y 435.097,Z 608.291,A -85,B 0,C 180,E1 -9609.688,E2 -9609.688} C_VEL
LIN {X 0,Y 434.673,Z 622.239,A -85,B 0,C 180,E1 -9611.648,E2 -9611.648} C_VEL
LIN {X 0,Y 437.465,Z 640.916,A -85,B 0,C 180,E1 -9612.094,E2 -9612.094} C_VEL
LIN {X 0,Y 436.52,Z 732.705,A -85,B 0,C 180,E1 -9613.635,E2 -9613.635} C_VEL
LIN {X 0,Y 436.482,Z 735.621,A -85,B 0,C 180,E1 -9613.704,E2 -9613.704} C_VEL
LIN {X 0,Y 436.004,Z 739.468,A -85,B 0,C 180,E1 -9613.8,E2 -9613.8} C_VEL
LIN {X 0,Y 433.836,Z 746.961,A -85,B 0,C 180,E1 -9613.985,E2 -9613.985} C_VEL
LIN {X 0,Y 429.872,Z 757.867,A -85,B 0,C 180,E1 -9614.353,E2 -9614.353} C_VEL
LIN {X 0,Y 428.675,Z 763.273,A -85,B 0,C 180,E1 -9614.626,E2 -9614.626} C_VEL
LIN {X 0,Y 428.515,Z 765.022,A -85,B 0,C 180,E1 -9614.734,E2 -9614.734} C_VEL
LIN {X 0,Y 427.883,Z 775.635,A -85,B 0,C 180,E1 -9615.493,E2 -9615.493} C_VEL
LIN {X 0,Y 427.28,Z 786.872,A -85,B 0,C 180,E1 -9616.519,E2 -9616.519} C_VEL
LIN {X 0,Y 426.557,Z 796.675,A -85,B 0,C 180,E1 -9617.631,E2 -9617.631} C_VEL
LIN {X 0,Y 425.974,Z 805.226,A -85,B 0,C 180,E1 -9618.821,E2 -9618.821} C_VEL
LIN {X 0,Y 425.367,Z 813.56,A -85,B 0,C 180,E1 -9620.249,E2 -9620.249} C_VEL
LIN {X 0,Y 424.818,Z 821.206,A -85,B 0,C 180,E1 -9621.916,E2 -9621.916} C_VEL
LIN {X 0,Y 424.569,Z 827.189,A -85,B 0,C 180,E1 -9623.627,E2 -9623.627} C_VEL
LIN {X 0,Y 424.274,Z 831.372,A -85,B 0,C 180,E1 -9625.248,E2 -9625.248} C_VEL
LIN {X 0,Y 424.216,Z 833.231,A -85,B 0,C 180,E1 -9626.2,E2 -9626.2} C_VEL
LIN {X 0,Y 424.236,Z 834.652,A -85,B 0,C 180,E1 -9627.151,E2 -9627.151} C_VEL
LIN {X 0,Y 424.092,Z 836.267,A -85,B 0,C 180,E1 -9629.05,E2 -9629.05} C_VEL
LIN {X 0,Y 424.085,Z 836.503,A -85,B 0,C 180,E1 -9629.999,E2 -9629.999} C_VEL
LIN {X 0,Y 424.091,Z 836.313,A -85,B 0,C 180,E1 -9630.949,E2 -9630.949} C_VEL
LIN {X 0,Y 424.235,Z 834.762,A -85,B 0,C 180,E1 -9632.848,E2 -9632.848} C_VEL
LIN {X 0,Y 424.215,Z 833.403,A -85,B 0,C 180,E1 -9633.799,E2 -9633.799} C_VEL
LIN {X 0,Y 424.365,Z 830.535,A -85,B 0,C 180,E1 -9635.225,E2 -9635.225} C_VEL
LIN {X 0,Y 424.541,Z 826.64,A -85,B 0,C 180,E1 -9636.654,E2 -9636.654} C_VEL
LIN {X 0,Y 424.807,Z 821.598,A -85,B 0,C 180,E1 -9638.083,E2 -9638.083} C_VEL
LIN {X 0,Y 425.256,Z 815.238,A -85,B 0,C 180,E1 -9639.512,E2 -9639.512} C_VEL
LIN {X 0,Y 425.819,Z 807.327,A -85,B 0,C 180,E1 -9640.94,E2 -9640.94} C_VEL
LIN {X 0,Y 426.362,Z 799.242,A -85,B 0,C 180,E1 -9642.131,E2 -9642.131} C_VEL
LIN {X 0,Y 427.121,Z 789.321,A -85,B 0,C 180,E1 -9643.317,E2 -9643.317} C_VEL
LIN {X 0,Y 427.761,Z 778.179,A -85,B 0,C 180,E1 -9644.388,E2 -9644.388} C_VEL
LIN {X 0,Y 428.418,Z 767.265,A -85,B 0,C 180,E1 -9645.216,E2 -9645.216} C_VEL
LIN {X 0,Y 428.987,Z 755.013,A -85,B 0,C 180,E1 -9645.926,E2 -9645.926} C_VEL
LIN {X 0,Y 429.519,Z 741.466,A -85,B 0,C 180,E1 -9646.485,E2 -9646.485} C_VEL
LIN {X 0,Y 429.781,Z 728.9,A -85,B 0,C 180,E1 -9646.811,E2 -9646.811} C_VEL
LIN {X 0,Y 430.614,Z 641.985,A -85,B 0,C 180,E1 -9648.278,E2 -9648.278} C_VEL
LIN {X 0,Y 427.405,Z 623.252,A -85,B 0,C 180,E1 -9648.751,E2 -9648.751} C_VEL
LIN {X 0,Y 427.86,Z 609.245,A -85,B 0,C 180,E1 -9650.974,E2 -9650.974} C_VEL
LIN {X 0,Y 428.668,Z 591.672,A -85,B 0,C 180,E1 -9653.913,E2 -9653.913} C_VEL
LIN {X 0,Y 429.532,Z 573.852,A -85,B 0,C 180,E1 -9657.002,E2 -9657.002} C_VEL
LIN {X 0,Y 429.71,Z 568.301,A -85,B 0,C 180,E1 -9657.971,E2 -9657.971} C_VEL
LIN {X 0,Y 427.9,Z 558.638,A -85,B 0,C 180,E1 -9659.789,E2 -9659.789} C_VEL
LIN {X 0,Y 425.324,Z 547.504,A -85,B 0,C 180,E1 -9661.92,E2 -9661.92} C_VEL
LIN {X 0,Y 425.297,Z 547.509,A -85,B 0,C 180,E1 -9665.334,E2 -9665.334} C_VEL
LIN {X 0,Y 425.299,Z 547.504,A -85,B 0,C 180,E1 -9669.043,E2 -9669.043} C_VEL
LIN {X 0,Y 425.273,Z 547.506,A -85,B 0,C 180,E1 -9672.651,E2 -9672.651} C_VEL
LIN {X 0,Y 425.313,Z 547.504,A -85,B 0,C 180,E1 -9676.05,E2 -9676.05} C_VEL
LIN {X 0,Y 425.304,Z 547.506,A -85,B 0,C 180,E1 -9678.625,E2 -9678.625} C_VEL
LIN {X 0,Y 425.339,Z 547.504,A -85,B 0,C 180,E1 -9680.083,E2 -9680.083} C_VEL
LIN {X 0,Y 430.061,Z 561.196,A -85,B 0,C 180,E1 -9680.546,E2 -9680.546} C_VEL
LIN {X 0,Y 429.238,Z 628.208,A -85,B 0,C 180,E1 -9681.803,E2 -9681.803} C_VEL
LIN {X 0,Y 429.166,Z 642.25,A -85,B 0,C 180,E1 -9682.278,E2 -9682.278} C_VEL
LIN {X 0,Y 428.893,Z 654.931,A -85,B 0,C 180,E1 -9682.906,E2 -9682.906} C_VEL
LIN {X 0,Y 428.525,Z 666.639,A -85,B 0,C 180,E1 -9683.681,E2 -9683.681} C_VEL
LIN {X 0,Y 428.035,Z 678.005,A -85,B 0,C 180,E1 -9684.635,E2 -9684.635} C_VEL
LIN {X 0,Y 427.511,Z 688.702,A -85,B 0,C 180,E1 -9685.767,E2 -9685.767} C_VEL
LIN {X 0,Y 426.984,Z 698.806,A -85,B 0,C 180,E1 -9687.1,E2 -9687.1} C_VEL
LIN {X 0,Y 426.558,Z 706.859,A -85,B 0,C 180,E1 -9688.415,E2 -9688.415} C_VEL
LIN {X 0,Y 426.13,Z 713.719,A -85,B 0,C 180,E1 -9689.799,E2 -9689.799} C_VEL
LIN {X 0,Y 425.759,Z 720.006,A -85,B 0,C 180,E1 -9691.399,E2 -9691.399} C_VEL
LIN {X 0,Y 425.561,Z 725.031,A -85,B 0,C 180,E1 -9693.096,E2 -9693.096} C_VEL
LIN {X 0,Y 425.349,Z 728.156,A -85,B 0,C 180,E1 -9694.558,E2 -9694.558} C_VEL
LIN {X 0,Y 425.259,Z 729.732,A -85,B 0,C 180,E1 -9695.596,E2 -9695.596} C_VEL
LIN {X 0,Y 425.23,Z 730.847,A -85,B 0,C 180,E1 -9696.63,E2 -9696.63} C_VEL
LIN {X 0,Y 425.256,Z 731.446,A -85,B 0,C 180,E1 -9697.737,E2 -9697.737} C_VEL
LIN {X 0,Y 425.296,Z 731.549,A -85,B 0,C 180,E1 -9698.682,E2 -9698.682} C_VEL
LIN {X 0,Y 425.403,Z 730.774,A -85,B 0,C 180,E1 -9700.332,E2 -9700.332} C_VEL
LIN {X 0,Y 425.585,Z 729.13,A -85,B 0,C 180,E1 -9701.714,E2 -9701.714} C_VEL
LIN {X 0,Y 425.826,Z 726.401,A -85,B 0,C 180,E1 -9703.181,E2 -9703.181} C_VEL
LIN {X 0,Y 426.169,Z 722.413,A -85,B 0,C 180,E1 -9704.701,E2 -9704.701} C_VEL
LIN {X 0,Y 426.67,Z 716.488,A -85,B 0,C 180,E1 -9706.362,E2 -9706.362} C_VEL
LIN {X 0,Y 427.172,Z 709.448,A -85,B 0,C 180,E1 -9707.891,E2 -9707.891} C_VEL
LIN {X 0,Y 427.698,Z 702.453,A -85,B 0,C 180,E1 -9709.107,E2 -9709.107} C_VEL
LIN {X 0,Y 428.293,Z 693.116,A -85,B 0,C 180,E1 -9710.425,E2 -9710.425} C_VEL
LIN {X 0,Y 428.907,Z 682.39,A -85,B 0,C 180,E1 -9711.638,E2 -9711.638} C_VEL
LIN {X 0,Y 429.468,Z 671.66,A -85,B 0,C 180,E1 -9712.596,E2 -9712.596} C_VEL
LIN {X 0,Y 429.919,Z 659.751,A -85,B 0,C 180,E1 -9713.429,E2 -9713.429} C_VEL
LIN {X 0,Y 430.208,Z 647.461,A -85,B 0,C 180,E1 -9714.081,E2 -9714.081} C_VEL
LIN {X 0,Y 430.281,Z 634.112,A -85,B 0,C 180,E1 -9714.57,E2 -9714.57} C_VEL
LIN {X 0,Y 430.347,Z 615.203,A -85,B 0,C 180,E1 -9714.978,E2 -9714.978} C_VEL
LIN {X 0,Y 431.194,Z 561.915,A -85,B 0,C 180,E1 -9716.014,E2 -9716.014} C_VEL
LIN {X 0,Y 425.499,Z 547.869,A -85,B 0,C 180,E1 -9716.627,E2 -9716.627} C_VEL
LIN {X 0,Y 425.442,Z 547.492,A -85,B 0,C 180,E1 -9716.685,E2 -9716.685} C_VEL
LIN {X 0,Y 425.694,Z 547.461,A -85,B 0,C 180,E1 -9720,E2 -9720} C_VEL
LIN {X 0,Y 425.549,Z 547.479,A -85,B 0,C 180,E1 -9722.84,E2 -9722.84} C_VEL
LIN {X 0,Y 425.569,Z 547.472,A -85,B 0,C 180,E1 -9725.687,E2 -9725.687} C_VEL
LIN {X 0,Y 425.432,Z 547.492,A -85,B 0,C 180,E1 -9728.55,E2 -9728.55} C_VEL
LIN {X 0,Y 425.419,Z 547.492,A -85,B 0,C 180,E1 -9732.402,E2 -9732.402} C_VEL
LIN {X 0,Y 425.378,Z 547.493,A -85,B 0,C 180,E1 -9736.312,E2 -9736.312} C_VEL
LIN {X 0,Y 425.318,Z 547.502,A -85,B 0,C 180,E1 -9739.636,E2 -9739.636} C_VEL
LIN {X 0,Y 425.297,Z 547.507,A -85,B 0,C 180,E1 -9743.366,E2 -9743.366} C_VEL
LIN {X 0,Y 425.339,Z 547.505,A -85,B 0,C 180,E1 -9746.845,E2 -9746.845} C_VEL
LIN {X 0,Y 425.309,Z 547.504,A -85,B 0,C 180,E1 -9749.718,E2 -9749.718} C_VEL
LIN {X 0,Y 425.274,Z 547.513,A -85,B 0,C 180,E1 -9753.049,E2 -9753.049} C_VEL
LIN {X 0,Y 425.277,Z 547.509,A -85,B 0,C 180,E1 -9755.93,E2 -9755.93} C_VEL
LIN {X 0,Y 425.307,Z 547.509,A -85,B 0,C 180,E1 -9759.047,E2 -9759.047} C_VEL
LIN {X 0,Y 425.325,Z 547.505,A -85,B 0,C 180,E1 -9762.647,E2 -9762.647} C_VEL
LIN {X 0,Y 425.329,Z 547.504,A -85,B 0,C 180,E1 -9766.055,E2 -9766.055} C_VEL
LIN {X 0,Y 425.305,Z 547.509,A -85,B 0,C 180,E1 -9768.627,E2 -9768.627} C_VEL
LIN {X 0,Y 425.32,Z 547.508,A -85,B 0,C 180,E1 -9771.105,E2 -9771.105} C_VEL
LIN {X 0,Y 425.297,Z 547.513,A -85,B 0,C 180,E1 -9774.665,E2 -9774.665} C_VEL
LIN {X 0,Y 425.289,Z 547.527,A -85,B 0,C 180,E1 -9777.58,E2 -9777.58} C_VEL
LIN {X 0,Y 428.4,Z 560.101,A -85,B 0,C 180,E1 -9779.946,E2 -9779.946} C_VEL
LIN {X 0,Y 430.116,Z 568.649,A -85,B 0,C 180,E1 -9781.451,E2 -9781.451} C_VEL
LIN {X 0,Y 429.712,Z 576.915,A -85,B 0,C 180,E1 -9782.747,E2 -9782.747} C_VEL
LIN {X 0,Y 428.313,Z 596.892,A -85,B 0,C 180,E1 -9785.783,E2 -9785.783} C_VEL
LIN {X 0,Y 427.191,Z 617.028,A -85,B 0,C 180,E1 -9788.782,E2 -9788.782} C_VEL
LIN {X 0,Y 426.513,Z 632.178,A -85,B 0,C 180,E1 -9791,E2 -9791} C_VEL
LIN {X 0,Y 429.208,Z 657.011,A -85,B 0,C 180,E1 -9791.639,E2 -9791.639} C_VEL
LIN {X 0,Y 430.293,Z 670.465,A -85,B 0,C 180,E1 -9791.956,E2 -9791.956} C_VEL
LIN {X 0,Y 429.191,Z 749.945,A -85,B 0,C 180,E1 -9793.41,E2 -9793.41} C_VEL
LIN {X 0,Y 428.901,Z 762.88,A -85,B 0,C 180,E1 -9793.704,E2 -9793.704} C_VEL
LIN {X 0,Y 428.434,Z 775.359,A -85,B 0,C 180,E1 -9794.175,E2 -9794.175} C_VEL
LIN {X 0,Y 427.929,Z 786.567,A -85,B 0,C 180,E1 -9794.766,E2 -9794.766} C_VEL
LIN {X 0,Y 427.305,Z 798.535,A -85,B 0,C 180,E1 -9795.597,E2 -9795.597} C_VEL
LIN {X 0,Y 426.719,Z 809.048,A -85,B 0,C 180,E1 -9796.536,E2 -9796.536} C_VEL
LIN {X 0,Y 426.071,Z 818.845,A -85,B 0,C 180,E1 -9797.619,E2 -9797.619} C_VEL
LIN {X 0,Y 425.446,Z 827.653,A -85,B 0,C 180,E1 -9798.809,E2 -9798.809} C_VEL
LIN {X 0,Y 425.05,Z 834.906,A -85,B 0,C 180,E1 -9800.003,E2 -9800.003} C_VEL
LIN {X 0,Y 424.683,Z 842.011,A -85,B 0,C 180,E1 -9801.435,E2 -9801.435} C_VEL
LIN {X 0,Y 424.438,Z 847.652,A -85,B 0,C 180,E1 -9802.867,E2 -9802.867} C_VEL
LIN {X 0,Y 424.291,Z 852.074,A -85,B 0,C 180,E1 -9804.297,E2 -9804.297} C_VEL
LIN {X 0,Y 424.287,Z 854.404,A -85,B 0,C 180,E1 -9805.25,E2 -9805.25} C_VEL
LIN {X 0,Y 424.205,Z 856.298,A -85,B 0,C 180,E1 -9806.201,E2 -9806.201} C_VEL
LIN {X 0,Y 424.242,Z 857.73,A -85,B 0,C 180,E1 -9807.152,E2 -9807.152} C_VEL
LIN {X 0,Y 424.216,Z 858.738,A -85,B 0,C 180,E1 -9808.102,E2 -9808.102} C_VEL
LIN {X 0,Y 424.206,Z 859.354,A -85,B 0,C 180,E1 -9809.052,E2 -9809.052} C_VEL
LIN {X 0,Y 424.218,Z 859.575,A -85,B 0,C 180,E1 -9810.001,E2 -9810.001} C_VEL
LIN {X 0,Y 424.211,Z 858.734,A -85,B 0,C 180,E1 -9811.9,E2 -9811.9} C_VEL
LIN {X 0,Y 424.231,Z 857.724,A -85,B 0,C 180,E1 -9812.849,E2 -9812.849} C_VEL
LIN {X 0,Y 424.189,Z 856.289,A -85,B 0,C 180,E1 -9813.801,E2 -9813.801} C_VEL
LIN {X 0,Y 424.299,Z 853.307,A -85,B 0,C 180,E1 -9815.228,E2 -9815.228} C_VEL
LIN {X 0,Y 424.395,Z 849.256,A -85,B 0,C 180,E1 -9816.657,E2 -9816.657} C_VEL
LIN {X 0,Y 424.617,Z 842.999,A -85,B 0,C 180,E1 -9818.328,E2 -9818.328} C_VEL
LIN {X 0,Y 424.96,Z 836.172,A -85,B 0,C 180,E1 -9819.76,E2 -9819.76} C_VEL
LIN {X 0,Y 425.34,Z 829.193,A -85,B 0,C 180,E1 -9820.954,E2 -9820.954} C_VEL
LIN {X 0,Y 425.904,Z 820.758,A -85,B 0,C 180,E1 -9822.146,E2 -9822.146} C_VEL
LIN {X 0,Y 426.58,Z 810.294,A -85,B 0,C 180,E1 -9823.336,E2 -9823.336} C_VEL
LIN {X 0,Y 427.156,Z 799.911,A -85,B 0,C 180,E1 -9824.289,E2 -9824.289} C_VEL
LIN {X 0,Y 427.812,Z 788.46,A -85,B 0,C 180,E1 -9825.118,E2 -9825.118} C_VEL
LIN {X 0,Y 428.411,Z 776.545,A -85,B 0,C 180,E1 -9825.766,E2 -9825.766} C_VEL
LIN {X 0,Y 428.862,Z 763.631,A -85,B 0,C 180,E1 -9826.268,E2 -9826.268} C_VEL
LIN {X 0,Y 429.114,Z 751.4,A -85,B 0,C 180,E1 -9826.564,E2 -9826.564} C_VEL
LIN {X 0,Y 429.885,Z 669.576,A -85,B 0,C 180,E1 -9827.928,E2 -9827.928} C_VEL
LIN {X 0,Y 426.271,Z 637.652,A -85,B 0,C 180,E1 -9828.692,E2 -9828.692} C_VEL
LIN {X 0,Y 427.424,Z 614.641,A -85,B 0,C 180,E1 -9832.433,E2 -9832.433} C_VEL
LIN {X 0,Y 428.721,Z 591.348,A -85,B 0,C 180,E1 -9836.271,E2 -9836.271} C_VEL
LIN {X 0,Y 430.076,Z 571.045,A -85,B 0,C 180,E1 -9839.667,E2 -9839.667} C_VEL
LIN {X 0,Y 429.592,Z 566.518,A -85,B 0,C 180,E1 -9840.475,E2 -9840.475} C_VEL
LIN {X 0,Y 426.283,Z 551.848,A -85,B 0,C 180,E1 -9843.243,E2 -9843.243} C_VEL
LIN {X 0,Y 425.328,Z 547.505,A -85,B 0,C 180,E1 -9844.11,E2 -9844.11} C_VEL
LIN {X 0,Y 425.282,Z 547.509,A -85,B 0,C 180,E1 -9847.694,E2 -9847.694} C_VEL
LIN {X 0,Y 425.283,Z 547.509,A -85,B 0,C 180,E1 -9850.521,E2 -9850.521} C_VEL
LIN {X 0,Y 425.259,Z 547.507,A -85,B 0,C 180,E1 -9853.351,E2 -9853.351} C_VEL
LIN {X 0,Y 425.266,Z 547.511,A -85,B 0,C 180,E1 -9856.648,E2 -9856.648} C_VEL
LIN {X 0,Y 425.288,Z 547.507,A -85,B 0,C 180,E1 -9859.873,E2 -9859.873} C_VEL
LIN {X 0,Y 425.286,Z 547.504,A -85,B 0,C 180,E1 -9862.487,E2 -9862.487} C_VEL
LIN {X 0,Y 425.309,Z 547.505,A -85,B 0,C 180,E1 -9865.817,E2 -9865.817} C_VEL
LIN {X 0,Y 425.291,Z 547.5,A -85,B 0,C 180,E1 -9869.239,E2 -9869.239} C_VEL
LIN {X 0,Y 425.349,Z 547.498,A -85,B 0,C 180,E1 -9872.442,E2 -9872.442} C_VEL
LIN {X 0,Y 425.351,Z 547.491,A -85,B 0,C 180,E1 -9875.602,E2 -9875.602} C_VEL
LIN {X 0,Y 425.293,Z 547.506,A -85,B 0,C 180,E1 -9878.681,E2 -9878.681} C_VEL
LIN {X 0,Y 425.333,Z 547.489,A -85,B 0,C 180,E1 -9881.703,E2 -9881.703} C_VEL
LIN {X 0,Y 425.349,Z 547.496,A -85,B 0,C 180,E1 -9884.671,E2 -9884.671} C_VEL
LIN {X 0,Y 425.412,Z 547.489,A -85,B 0,C 180,E1 -9887.598,E2 -9887.598} C_VEL
LIN {X 0,Y 425.443,Z 547.483,A -85,B 0,C 180,E1 -9891.45,E2 -9891.45} C_VEL
LIN {X 0,Y 425.554,Z 547.472,A -85,B 0,C 180,E1 -9894.313,E2 -9894.313} C_VEL
LIN {X 0,Y 425.573,Z 547.464,A -85,B 0,C 180,E1 -9898.107,E2 -9898.107} C_VEL
LIN {X 0,Y 425.701,Z 547.458,A -85,B 0,C 180,E1 -9900,E2 -9900} C_VEL
LIN {X 0,Y 425.547,Z 547.471,A -85,B 0,C 180,E1 -9902.84,E2 -9902.84} C_VEL
LIN {X 0,Y 425.53,Z 547.471,A -85,B 0,C 180,E1 -9906.639,E2 -9906.639} C_VEL
LIN {X 0,Y 425.401,Z 547.496,A -85,B 0,C 180,E1 -9909.509,E2 -9909.509} C_VEL
LIN {X 0,Y 425.394,Z 547.48,A -85,B 0,C 180,E1 -9912.904,E2 -9912.904} C_VEL
LIN {X 0,Y 425.362,Z 547.496,A -85,B 0,C 180,E1 -9916.605,E2 -9916.605} C_VEL
LIN {X 0,Y 425.329,Z 547.492,A -85,B 0,C 180,E1 -9919.636,E2 -9919.636} C_VEL
LIN {X 0,Y 425.308,Z 547.504,A -85,B 0,C 180,E1 -9923.365,E2 -9923.365} C_VEL
LIN {X 0,Y 425.348,Z 547.497,A -85,B 0,C 180,E1 -9926.844,E2 -9926.844} C_VEL
LIN {X 0,Y 425.292,Z 547.508,A -85,B 0,C 180,E1 -9929.72,E2 -9929.72} C_VEL
LIN {X 0,Y 425.283,Z 547.508,A -85,B 0,C 180,E1 -9933.048,E2 -9933.048} C_VEL
LIN {X 0,Y 425.283,Z 547.506,A -85,B 0,C 180,E1 -9935.929,E2 -9935.929} C_VEL
LIN {X 0,Y 425.295,Z 547.504,A -85,B 0,C 180,E1 -9939.043,E2 -9939.043} C_VEL
LIN {X 0,Y 425.276,Z 547.506,A -85,B 0,C 180,E1 -9942.653,E2 -9942.653} C_VEL
LIN {X 0,Y 425.263,Z 547.508,A -85,B 0,C 180,E1 -9946.044,E2 -9946.044} C_VEL
LIN {X 0,Y 425.284,Z 547.508,A -85,B 0,C 180,E1 -9949.48,E2 -9949.48} C_VEL
LIN {X 0,Y 425.281,Z 547.503,A -85,B 0,C 180,E1 -9952.488,E2 -9952.488} C_VEL
LIN {X 0,Y 425.311,Z 547.508,A -85,B 0,C 180,E1 -9955.817,E2 -9955.817} C_VEL
LIN {X 0,Y 425.324,Z 547.511,A -85,B 0,C 180,E1 -9959.489,E2 -9959.489} C_VEL
LIN {X 0,Y 425.348,Z 547.764,A -85,B 0,C 180,E1 -9959.738,E2 -9959.738} C_VEL
LIN {X 0,Y 428.517,Z 561.034,A -85,B 0,C 180,E1 -9962.014,E2 -9962.014} C_VEL
LIN {X 0,Y 430.078,Z 568.591,A -85,B 0,C 180,E1 -9963.295,E2 -9963.295} C_VEL
LIN {X 0,Y 429.777,Z 577.19,A -85,B 0,C 180,E1 -9964.631,E2 -9964.631} C_VEL
LIN {X 0,Y 428.738,Z 596.589,A -85,B 0,C 180,E1 -9967.596,E2 -9967.596} C_VEL
LIN {X 0,Y 428.048,Z 615.111,A -85,B 0,C 180,E1 -9970.331,E2 -9970.331} C_VEL
LIN {X 0,Y 427.805,Z 622.442,A -85,B 0,C 180,E1 -9971.351,E2 -9971.351} C_VEL
LIN {X 0,Y 430.699,Z 641.012,A -85,B 0,C 180,E1 -9971.803,E2 -9971.803} C_VEL
LIN {X 0,Y 429.732,Z 732.827,A -85,B 0,C 180,E1 -9973.369,E2 -9973.369} C_VEL
LIN {X 0,Y 429.333,Z 746.322,A -85,B 0,C 180,E1 -9973.781,E2 -9973.781} C_VEL
LIN {X 0,Y 428.762,Z 758.892,A -85,B 0,C 180,E1 -9974.369,E2 -9974.369} C_VEL
LIN {X 0,Y 428.515,Z 765.022,A -85,B 0,C 180,E1 -9974.734,E2 -9974.734} C_VEL
LIN {X 0,Y 427.62,Z 770.325,A -85,B 0,C 180,E1 -9975.064,E2 -9975.064} C_VEL
LIN {X 0,Y 424.391,Z 778.754,A -85,B 0,C 180,E1 -9975.619,E2 -9975.619} C_VEL
LIN {X 0,Y 421.083,Z 786.741,A -85,B 0,C 180,E1 -9976.275,E2 -9976.275} C_VEL
LIN {X 0,Y 420.072,Z 791.348,A -85,B 0,C 180,E1 -9976.758,E2 -9976.758} C_VEL
LIN {X 0,Y 419.347,Z 800.487,A -85,B 0,C 180,E1 -9977.907,E2 -9977.907} C_VEL
LIN {X 0,Y 418.645,Z 809.831,A -85,B 0,C 180,E1 -9979.358,E2 -9979.358} C_VEL
LIN {X 0,Y 418.092,Z 817.263,A -85,B 0,C 180,E1 -9980.81,E2 -9980.81} C_VEL
LIN {X 0,Y 417.653,Z 823.234,A -85,B 0,C 180,E1 -9982.263,E2 -9982.263} C_VEL
LIN {X 0,Y 417.48,Z 827.666,A -85,B 0,C 180,E1 -9983.617,E2 -9983.617} C_VEL
LIN {X 0,Y 417.213,Z 831.565,A -85,B 0,C 180,E1 -9985.168,E2 -9985.168} C_VEL
LIN {X 0,Y 417.124,Z 833.425,A -85,B 0,C 180,E1 -9986.135,E2 -9986.135} C_VEL
LIN {X 0,Y 417.152,Z 834.845,A -85,B 0,C 180,E1 -9987.102,E2 -9987.102} C_VEL
LIN {X 0,Y 417.014,Z 836.459,A -85,B 0,C 180,E1 -9989.034,E2 -9989.034} C_VEL
LIN {X 0,Y 417.004,Z 836.695,A -85,B 0,C 180,E1 -9989.999,E2 -9989.999} C_VEL
LIN {X 0,Y 417.081,Z 835.92,A -85,B 0,C 180,E1 -9991.93,E2 -9991.93} C_VEL
LIN {X 0,Y 417.137,Z 834.955,A -85,B 0,C 180,E1 -9992.896,E2 -9992.896} C_VEL
LIN {X 0,Y 417.123,Z 833.595,A -85,B 0,C 180,E1 -9993.864,E2 -9993.864} C_VEL
LIN {X 0,Y 417.312,Z 830.726,A -85,B 0,C 180,E1 -9995.314,E2 -9995.314} C_VEL
LIN {X 0,Y 417.479,Z 826.83,A -85,B 0,C 180,E1 -9996.767,E2 -9996.767} C_VEL
LIN {X 0,Y 417.778,Z 821.786,A -85,B 0,C 180,E1 -9998.22,E2 -9998.22} C_VEL
LIN {X 0,Y 418.245,Z 815.425,A -85,B 0,C 180,E1 -9999.673,E2 -9999.673} C_VEL
LIN {X 0,Y 418.836,Z 807.512,A -85,B 0,C 180,E1 -10001.125,E2 -10001.125} C_VEL
LIN {X 0,Y 419.431,Z 799.424,A -85,B 0,C 180,E1 -10002.335,E2 -10002.335} C_VEL
LIN {X 0,Y 420.224,Z 789.498,A -85,B 0,C 180,E1 -10003.54,E2 -10003.54} C_VEL
LIN {X 0,Y 420.885,Z 778.351,A -85,B 0,C 180,E1 -10004.628,E2 -10004.628} C_VEL
LIN {X 0,Y 421.588,Z 767.429,A -85,B 0,C 180,E1 -10005.468,E2 -10005.468} C_VEL
LIN {X 0,Y 422.179,Z 755.161,A -85,B 0,C 180,E1 -10006.19,E2 -10006.19} C_VEL
LIN {X 0,Y 422.723,Z 741.592,A -85,B 0,C 180,E1 -10006.758,E2 -10006.758} C_VEL
LIN {X 0,Y 423.001,Z 728.956,A -85,B 0,C 180,E1 -10007.089,E2 -10007.089} C_VEL
LIN {X 0,Y 423.908,Z 643.001,A -85,B 0,C 180,E1 -10008.561,E2 -10008.561} C_VEL
LIN {X 0,Y 420.546,Z 623.29,A -85,B 0,C 180,E1 -10009.079,E2 -10009.079} C_VEL
LIN {X 0,Y 421.219,Z 604.863,A -85,B 0,C 180,E1 -10012.048,E2 -10012.048} C_VEL
LIN {X 0,Y 422.089,Z 586.974,A -85,B 0,C 180,E1 -10015.123,E2 -10015.123} C_VEL
LIN {X 0,Y 422.898,Z 570.229,A -85,B 0,C 180,E1 -10018.054,E2 -10018.054} C_VEL
LIN {X 0,Y 421.191,Z 560.981,A -85,B 0,C 180,E1 -10019.81,E2 -10019.81} C_VEL
LIN {X 0,Y 418.258,Z 548.386,A -85,B 0,C 180,E1 -10022.276,E2 -10022.276} C_VEL
LIN {X 0,Y 418.257,Z 548.39,A -85,B 0,C 180,E1 -10024.84,E2 -10024.84} C_VEL
LIN {X 0,Y 418.257,Z 548.387,A -85,B 0,C 180,E1 -10028.44,E2 -10028.44} C_VEL
LIN {X 0,Y 418.219,Z 548.39,A -85,B 0,C 180,E1 -10030.946,E2 -10030.946} C_VEL
LIN {X 0,Y 418.211,Z 548.379,A -85,B 0,C 180,E1 -10033.729,E2 -10033.729} C_VEL
LIN {X 0,Y 418.262,Z 548.382,A -85,B 0,C 180,E1 -10036.455,E2 -10036.455} C_VEL
LIN {X 0,Y 418.298,Z 548.382,A -85,B 0,C 180,E1 -10039.822,E2 -10039.822} C_VEL
LIN {X 0,Y 423.25,Z 562.718,A -85,B 0,C 180,E1 -10040.315,E2 -10040.315} C_VEL
LIN {X 0,Y 422.358,Z 629.243,A -85,B 0,C 180,E1 -10041.589,E2 -10041.589} C_VEL
LIN {X 0,Y 422.307,Z 643.335,A -85,B 0,C 180,E1 -10042.076,E2 -10042.076} C_VEL
LIN {X 0,Y 422.028,Z 655.745,A -85,B 0,C 180,E1 -10042.701,E2 -10042.701} C_VEL
LIN {X 0,Y 421.577,Z 668.506,A -85,B 0,C 180,E1 -10043.566,E2 -10043.566} C_VEL
LIN {X 0,Y 421.122,Z 678.776,A -85,B 0,C 180,E1 -10044.449,E2 -10044.449} C_VEL
LIN {X 0,Y 420.645,Z 688.948,A -85,B 0,C 180,E1 -10045.53,E2 -10045.53} C_VEL
LIN {X 0,Y 420.048,Z 699.111,A -85,B 0,C 180,E1 -10046.873,E2 -10046.873} C_VEL
LIN {X 0,Y 419.614,Z 707.015,A -85,B 0,C 180,E1 -10048.157,E2 -10048.157} C_VEL
LIN {X 0,Y 419.203,Z 713.899,A -85,B 0,C 180,E1 -10049.526,E2 -10049.526} C_VEL
LIN {X 0,Y 418.821,Z 719.427,A -85,B 0,C 180,E1 -10050.88,E2 -10050.88} C_VEL
LIN {X 0,Y 418.612,Z 724.469,A -85,B 0,C 180,E1 -10052.466,E2 -10052.466} C_VEL
LIN {X 0,Y 418.37,Z 728.33,A -85,B 0,C 180,E1 -10054.102,E2 -10054.102} C_VEL
LIN {X 0,Y 418.28,Z 730.177,A -85,B 0,C 180,E1 -10055.162,E2 -10055.162} C_VEL
LIN {X 0,Y 418.211,Z 731.452,A -85,B 0,C 180,E1 -10056.214,E2 -10056.214} C_VEL
LIN {X 0,Y 418.237,Z 732.408,A -85,B 0,C 180,E1 -10057.546,E2 -10057.546} C_VEL
LIN {X 0,Y 418.313,Z 732.435,A -85,B 0,C 180,E1 -10059.34,E2 -10059.34} C_VEL
LIN {X 0,Y 418.401,Z 731.841,A -85,B 0,C 180,E1 -10060.37,E2 -10060.37} C_VEL
LIN {X 0,Y 418.533,Z 730.746,A -85,B 0,C 180,E1 -10061.395,E2 -10061.395} C_VEL
LIN {X 0,Y 418.808,Z 727.999,A -85,B 0,C 180,E1 -10063.035,E2 -10063.035} C_VEL
LIN {X 0,Y 419.087,Z 724.622,A -85,B 0,C 180,E1 -10064.436,E2 -10064.436} C_VEL
LIN {X 0,Y 419.543,Z 719.832,A -85,B 0,C 180,E1 -10065.933,E2 -10065.933} C_VEL
LIN {X 0,Y 420.081,Z 713.658,A -85,B 0,C 180,E1 -10067.438,E2 -10067.438} C_VEL
LIN {X 0,Y 420.649,Z 705.932,A -85,B 0,C 180,E1 -10068.922,E2 -10068.922} C_VEL
LIN {X 0,Y 421.272,Z 697.903,A -85,B 0,C 180,E1 -10070.162,E2 -10070.162} C_VEL
LIN {X 0,Y 421.905,Z 688.241,A -85,B 0,C 180,E1 -10071.378,E2 -10071.378} C_VEL
LIN {X 0,Y 422.45,Z 678.696,A -85,B 0,C 180,E1 -10072.352,E2 -10072.352} C_VEL
LIN {X 0,Y 422.967,Z 666.705,A -85,B 0,C 180,E1 -10073.321,E2 -10073.321} C_VEL
LIN {X 0,Y 423.418,Z 653.951,A -85,B 0,C 180,E1 -10074.105,E2 -10074.105} C_VEL
LIN {X 0,Y 423.593,Z 641.009,A -85,B 0,C 180,E1 -10074.675,E2 -10074.675} C_VEL
LIN {X 0,Y 423.641,Z 628.122,A -85,B 0,C 180,E1 -10075.046,E2 -10075.046} C_VEL
LIN {X 0,Y 424.613,Z 563.683,A -85,B 0,C 180,E1 -10076.335,E2 -10076.335} C_VEL
LIN {X 0,Y 418.59,Z 549.006,A -85,B 0,C 180,E1 -10077.004,E2 -10077.004} C_VEL
LIN {X 0,Y 418.506,Z 548.356,A -85,B 0,C 180,E1 -10077.058,E2 -10077.058} C_VEL
LIN {X 0,Y 418.663,Z 548.337,A -85,B 0,C 180,E1 -10080,E2 -10080} C_VEL
LIN {X 0,Y 418.503,Z 548.356,A -85,B 0,C 180,E1 -10082.888,E2 -10082.888} C_VEL
LIN {X 0,Y 418.524,Z 548.349,A -85,B 0,C 180,E1 -10085.783,E2 -10085.783} C_VEL
LIN {X 0,Y 418.39,Z 548.371,A -85,B 0,C 180,E1 -10088.695,E2 -10088.695} C_VEL
LIN {X 0,Y 418.322,Z 548.375,A -85,B 0,C 180,E1 -10091.631,E2 -10091.631} C_VEL
LIN {X 0,Y 418.296,Z 548.383,A -85,B 0,C 180,E1 -10094.597,E2 -10094.597} C_VEL
LIN {X 0,Y 418.277,Z 548.38,A -85,B 0,C 180,E1 -10097.604,E2 -10097.604} C_VEL
LIN {X 0,Y 418.24,Z 548.39,A -85,B 0,C 180,E1 -10100.664,E2 -10100.664} C_VEL
LIN {X 0,Y 418.278,Z 548.38,A -85,B 0,C 180,E1 -10103.782,E2 -10103.782} C_VEL
LIN {X 0,Y 418.301,Z 548.379,A -85,B 0,C 180,E1 -10107.071,E2 -10107.071} C_VEL
LIN {X 0,Y 418.252,Z 548.385,A -85,B 0,C 180,E1 -10110.272,E2 -10110.272} C_VEL
LIN {X 0,Y 418.24,Z 548.385,A -85,B 0,C 180,E1 -10113.678,E2 -10113.678} C_VEL
LIN {X 0,Y 418.24,Z 548.384,A -85,B 0,C 180,E1 -10117.224,E2 -10117.224} C_VEL
LIN {X 0,Y 418.26,Z 548.382,A -85,B 0,C 180,E1 -10119.681,E2 -10119.681} C_VEL
LIN {X 0,Y 418.279,Z 548.384,A -85,B 0,C 180,E1 -10122.331,E2 -10122.331} C_VEL
LIN {X 0,Y 418.268,Z 548.384,A -85,B 0,C 180,E1 -10125.115,E2 -10125.115} C_VEL
LIN {X 0,Y 418.287,Z 548.381,A -85,B 0,C 180,E1 -10127.775,E2 -10127.775} C_VEL
LIN {X 0,Y 418.263,Z 548.385,A -85,B 0,C 180,E1 -10131.561,E2 -10131.561} C_VEL
LIN {X 0,Y 418.256,Z 548.391,A -85,B 0,C 180,E1 -10135.16,E2 -10135.16} C_VEL
LIN {X 0,Y 418.25,Z 548.54,A -85,B 0,C 180,E1 -10137.197,E2 -10137.197} C_VEL
LIN {X 0,Y 421.511,Z 561.507,A -85,B 0,C 180,E1 -10139.712,E2 -10139.712} C_VEL
LIN {X 0,Y 423.195,Z 569.744,A -85,B 0,C 180,E1 -10141.211,E2 -10141.211} C_VEL
LIN {X 0,Y 423.171,Z 574.279,A -85,B 0,C 180,E1 -10141.95,E2 -10141.95} C_VEL
LIN {X 0,Y 421.653,Z 594.493,A -85,B 0,C 180,E1 -10145.112,E2 -10145.112} C_VEL
LIN {X 0,Y 420.221,Z 617.918,A -85,B 0,C 180,E1 -10148.67,E2 -10148.67} C_VEL
LIN {X 0,Y 419.589,Z 630.952,A -85,B 0,C 180,E1 -10150.621,E2 -10150.621} C_VEL
LIN {X 0,Y 422.399,Z 655.982,A -85,B 0,C 180,E1 -10151.29,E2 -10151.29} C_VEL
LIN {X 0,Y 423.591,Z 670.676,A -85,B 0,C 180,E1 -10151.644,E2 -10151.644} C_VEL
LIN {X 0,Y 422.239,Z 758.419,A -85,B 0,C 180,E1 -10153.316,E2 -10153.316} C_VEL
LIN {X 0,Y 421.75,Z 771.827,A -85,B 0,C 180,E1 -10153.762,E2 -10153.762} C_VEL
LIN {X 0,Y 421.171,Z 784.429,A -85,B 0,C 180,E1 -10154.392,E2 -10154.392} C_VEL
LIN {X 0,Y 420.496,Z 796.8,A -85,B 0,C 180,E1 -10155.234,E2 -10155.234} C_VEL
LIN {X 0,Y 419.848,Z 807.198,A -85,B 0,C 180,E1 -10156.141,E2 -10156.141} C_VEL
LIN {X 0,Y 419.253,Z 816.712,A -85,B 0,C 180,E1 -10157.168,E2 -10157.168} C_VEL
LIN {X 0,Y 418.608,Z 825.841,A -85,B 0,C 180,E1 -10158.378,E2 -10158.378} C_VEL
LIN {X 0,Y 418.044,Z 834.719,A -85,B 0,C 180,E1 -10159.834,E2 -10159.834} C_VEL
LIN {X 0,Y 417.649,Z 841.822,A -85,B 0,C 180,E1 -10161.29,E2 -10161.29} C_VEL
LIN {X 0,Y 417.363,Z 847.461,A -85,B 0,C 180,E1 -10162.745,E2 -10162.745} C_VEL
LIN {X 0,Y 417.199,Z 851.882,A -85,B 0,C 180,E1 -10164.2,E2 -10164.2} C_VEL
LIN {X 0,Y 417.215,Z 854.212,A -85,B 0,C 180,E1 -10165.169,E2 -10165.169} C_VEL
LIN {X 0,Y 417.115,Z 856.106,A -85,B 0,C 180,E1 -10166.136,E2 -10166.136} C_VEL
LIN {X 0,Y 417.139,Z 857.538,A -85,B 0,C 180,E1 -10167.104,E2 -10167.104} C_VEL
LIN {X 0,Y 417.14,Z 858.546,A -85,B 0,C 180,E1 -10168.07,E2 -10168.07} C_VEL
LIN {X 0,Y 417.122,Z 859.162,A -85,B 0,C 180,E1 -10169.035,E2 -10169.035} C_VEL
LIN {X 0,Y 417.131,Z 859.382,A -85,B 0,C 180,E1 -10170.001,E2 -10170.001} C_VEL
LIN {X 0,Y 417.135,Z 858.542,A -85,B 0,C 180,E1 -10171.932,E2 -10171.932} C_VEL
LIN {X 0,Y 417.127,Z 857.531,A -85,B 0,C 180,E1 -10172.898,E2 -10172.898} C_VEL
LIN {X 0,Y 417.1,Z 856.095,A -85,B 0,C 180,E1 -10173.865,E2 -10173.865} C_VEL
LIN {X 0,Y 417.212,Z 853.114,A -85,B 0,C 180,E1 -10175.317,E2 -10175.317} C_VEL
LIN {X 0,Y 417.319,Z 849.063,A -85,B 0,C 180,E1 -10176.771,E2 -10176.771} C_VEL
LIN {X 0,Y 417.546,Z 842.806,A -85,B 0,C 180,E1 -10178.47,E2 -10178.47} C_VEL
LIN {X 0,Y 417.921,Z 835.981,A -85,B 0,C 180,E1 -10179.926,E2 -10179.926} C_VEL
LIN {X 0,Y 418.344,Z 829.003,A -85,B 0,C 180,E1 -10181.14,E2 -10181.14} C_VEL
LIN {X 0,Y 418.939,Z 820.57,A -85,B 0,C 180,E1 -10182.351,E2 -10182.351} C_VEL
LIN {X 0,Y 419.638,Z 810.109,A -85,B 0,C 180,E1 -10183.561,E2 -10183.561} C_VEL
LIN {X 0,Y 420.254,Z 799.73,A -85,B 0,C 180,E1 -10184.528,E2 -10184.528} C_VEL
LIN {X 0,Y 420.948,Z 788.286,A -85,B 0,C 180,E1 -10185.37,E2 -10185.37} C_VEL
LIN {X 0,Y 421.558,Z 776.381,A -85,B 0,C 180,E1 -10186.029,E2 -10186.029} C_VEL
LIN {X 0,Y 422.06,Z 763.488,A -85,B 0,C 180,E1 -10186.538,E2 -10186.538} C_VEL
LIN {X 0,Y 422.316,Z 751.312,A -85,B 0,C 180,E1 -10186.839,E2 -10186.839} C_VEL
LIN {X 0,Y 423.211,Z 671.375,A -85,B 0,C 180,E1 -10188.188,E2 -10188.188} C_VEL
LIN {X 0,Y 419.279,Z 637.152,A -85,B 0,C 180,E1 -10188.984,E2 -10188.984} C_VEL
LIN {X 0,Y 419.273,Z 636.219,A -85,B 0,C 180,E1 -10189.079,E2 -10189.079} C_VEL
LIN {X 0,Y 420.421,Z 614.854,A -85,B 0,C 180,E1 -10192.612,E2 -10192.612} C_VEL
LIN {X 0,Y 421.789,Z 591.848,A -85,B 0,C 180,E1 -10196.469,E2 -10196.469} C_VEL
LIN {X 0,Y 423.097,Z 573.372,A -85,B 0,C 180,E1 -10199.616,E2 -10199.616} C_VEL
LIN {X 0,Y 423.018,Z 569.839,A -85,B 0,C 180,E1 -10200.239,E2 -10200.239} C_VEL
LIN {X 0,Y 419.682,Z 554.604,A -85,B 0,C 180,E1 -10203.144,E2 -10203.144} C_VEL
LIN {X 0,Y 418.274,Z 548.385,A -85,B 0,C 180,E1 -10204.374,E2 -10204.374} C_VEL
LIN {X 0,Y 418.231,Z 548.387,A -85,B 0,C 180,E1 -10207.834,E2 -10207.834} C_VEL
LIN {X 0,Y 418.225,Z 548.392,A -85,B 0,C 180,E1 -10210.948,E2 -10210.948} C_VEL
LIN {X 0,Y 418.211,Z 548.381,A -85,B 0,C 180,E1 -10213.729,E2 -10213.729} C_VEL
LIN {X 0,Y 418.218,Z 548.388,A -85,B 0,C 180,E1 -10216.45,E2 -10216.45} C_VEL
LIN {X 0,Y 418.225,Z 548.384,A -85,B 0,C 180,E1 -10219.13,E2 -10219.13} C_VEL
LIN {X 0,Y 418.235,Z 548.382,A -85,B 0,C 180,E1 -10222.166,E2 -10222.166} C_VEL
LIN {X 0,Y 418.267,Z 548.386,A -85,B 0,C 180,E1 -10225.42,E2 -10225.42} C_VEL
LIN {X 0,Y 418.212,Z 548.381,A -85,B 0,C 180,E1 -10228.604,E2 -10228.604} C_VEL
LIN {X 0,Y 418.292,Z 548.379,A -85,B 0,C 180,E1 -10231.937,E2 -10231.937} C_VEL
LIN {X 0,Y 418.291,Z 548.37,A -85,B 0,C 180,E1 -10235.163,E2 -10235.163} C_VEL
LIN {X 0,Y 418.234,Z 548.385,A -85,B 0,C 180,E1 -10238.304,E2 -10238.304} C_VEL
LIN {X 0,Y 418.284,Z 548.37,A -85,B 0,C 180,E1 -10241.383,E2 -10241.383} C_VEL
LIN {X 0,Y 418.303,Z 548.374,A -85,B 0,C 180,E1 -10244.406,E2 -10244.406} C_VEL
LIN {X 0,Y 418.356,Z 548.371,A -85,B 0,C 180,E1 -10247.386,E2 -10247.386} C_VEL
LIN {X 0,Y 418.341,Z 548.361,A -85,B 0,C 180,E1 -10250.329,E2 -10250.329} C_VEL
LIN {X 0,Y 418.493,Z 548.355,A -85,B 0,C 180,E1 -10253.249,E2 -10253.249} C_VEL
LIN {X 0,Y 418.34,Z 548.372,A -85,B 0,C 180,E1 -10255.182,E2 -10255.182} C_VEL
LIN {X 0,Y 418.542,Z 548.338,A -85,B 0,C 180,E1 -10258.075,E2 -10258.075} C_VEL
LIN {X 0,Y 418.67,Z 548.334,A -85,B 0,C 180,E1 -10260,E2 -10260} C_VEL
LIN {X 0,Y 418.502,Z 548.349,A -85,B 0,C 180,E1 -10262.888,E2 -10262.888} C_VEL
LIN {X 0,Y 418.493,Z 548.347,A -85,B 0,C 180,E1 -10266.751,E2 -10266.751} C_VEL
LIN {X 0,Y 418.357,Z 548.375,A -85,B 0,C 180,E1 -10269.671,E2 -10269.671} C_VEL
LIN {X 0,Y 418.347,Z 548.358,A -85,B 0,C 180,E1 -10273.001,E2 -10273.001} C_VEL
LIN {X 0,Y 418.313,Z 548.374,A -85,B 0,C 180,E1 -10276.736,E2 -10276.736} C_VEL
LIN {X 0,Y 418.271,Z 548.372,A -85,B 0,C 180,E1 -10279.79,E2 -10279.79} C_VEL
LIN {X 0,Y 418.239,Z 548.384,A -85,B 0,C 180,E1 -10282.736,E2 -10282.736} C_VEL
LIN {X 0,Y 418.271,Z 548.374,A -85,B 0,C 180,E1 -10285.904,E2 -10285.904} C_VEL
LIN {X 0,Y 418.266,Z 548.38,A -85,B 0,C 180,E1 -10289.162,E2 -10289.162} C_VEL
LIN {X 0,Y 418.259,Z 548.384,A -85,B 0,C 180,E1 -10292.844,E2 -10292.844} C_VEL
LIN {X 0,Y 418.246,Z 548.385,A -85,B 0,C 180,E1 -10296.238,E2 -10296.238} C_VEL
LIN {X 0,Y 418.25,Z 548.383,A -85,B 0,C 180,E1 -10299.682,E2 -10299.682} C_VEL
LIN {X 0,Y 418.231,Z 548.387,A -85,B 0,C 180,E1 -10302.321,E2 -10302.321} C_VEL
LIN {X 0,Y 418.238,Z 548.385,A -85,B 0,C 180,E1 -10305.109,E2 -10305.109} C_VEL
LIN {X 0,Y 418.236,Z 548.371,A -85,B 0,C 180,E1 -10307.766,E2 -10307.766} C_VEL
LIN {X 0,Y 418.261,Z 548.382,A -85,B 0,C 180,E1 -10310.618,E2 -10310.618} C_VEL
LIN {X 0,Y 418.246,Z 548.388,A -85,B 0,C 180,E1 -10313.976,E2 -10313.976} C_VEL
LIN {X 0,Y 418.261,Z 548.386,A -85,B 0,C 180,E1 -10317.156,E2 -10317.156} C_VEL
LIN {X 0,Y 418.264,Z 548.401,A -85,B 0,C 180,E1 -10319.364,E2 -10319.364} C_VEL
LIN {X 0,Y 421.867,Z 563.586,A -85,B 0,C 180,E1 -10322,E2 -10322} C_VEL
LIN {X 0,Y 423.359,Z 571.617,A -85,B 0,C 180,E1 -10323.37,E2 -10323.37} C_VEL
LIN {X 0,Y 422.131,Z 593.136,A -85,B 0,C 180,E1 -10326.708,E2 -10326.708} C_VEL
LIN {X 0,Y 421.272,Z 613.44,A -85,B 0,C 180,E1 -10329.746,E2 -10329.746} C_VEL
LIN {X 0,Y 420.979,Z 622.483,A -85,B 0,C 180,E1 -10331.028,E2 -10331.028} C_VEL
LIN {X 0,Y 423.942,Z 641.583,A -85,B 0,C 180,E1 -10331.511,E2 -10331.511} C_VEL
LIN {X 0,Y 422.956,Z 732.95,A -85,B 0,C 180,E1 -10333.094,E2 -10333.094} C_VEL
LIN {X 0,Y 422.541,Z 746.479,A -85,B 0,C 180,E1 -10333.513,E2 -10333.513} C_VEL
LIN {X 0,Y 421.928,Z 759.064,A -85,B 0,C 180,E1 -10334.109,E2 -10334.109} C_VEL
LIN {X 0,Y 421.271,Z 771.184,A -85,B 0,C 180,E1 -10334.89,E2 -10334.89} C_VEL
LIN {X 0,Y 420.684,Z 781.908,A -85,B 0,C 180,E1 -10335.783,E2 -10335.783} C_VEL
LIN {X 0,Y 420.072,Z 791.348,A -85,B 0,C 180,E1 -10336.758,E2 -10336.758} C_VEL
LIN {X 0,Y 419.064,Z 795.864,A -85,B 0,C 180,E1 -10337.274,E2 -10337.274} C_VEL
LIN {X 0,Y 415.721,Z 802.847,A -85,B 0,C 180,E1 -10338.126,E2 -10338.126} C_VEL
LIN {X 0,Y 412.401,Z 809.247,A -85,B 0,C 180,E1 -10339.06,E2 -10339.06} C_VEL
LIN {X 0,Y 411.435,Z 812.821,A -85,B 0,C 180,E1 -10339.697,E2 -10339.697} C_VEL
LIN {X 0,Y 410.909,Z 819.621,A -85,B 0,C 180,E1 -10341.144,E2 -10341.144} C_VEL
LIN {X 0,Y 410.515,Z 825.147,A -85,B 0,C 180,E1 -10342.622,E2 -10342.622} C_VEL
LIN {X 0,Y 410.329,Z 829.478,A -85,B 0,C 180,E1 -10344.101,E2 -10344.101} C_VEL
LIN {X 0,Y 410.155,Z 831.758,A -85,B 0,C 180,E1 -10345.084,E2 -10345.084} C_VEL
LIN {X 0,Y 410.037,Z 833.618,A -85,B 0,C 180,E1 -10346.068,E2 -10346.068} C_VEL
LIN {X 0,Y 410.053,Z 835.039,A -85,B 0,C 180,E1 -10347.052,E2 -10347.052} C_VEL
LIN {X 0,Y 410.012,Z 836.035,A -85,B 0,C 180,E1 -10348.035,E2 -10348.035} C_VEL
LIN {X 0,Y 409.927,Z 836.888,A -85,B 0,C 180,E1 -10349.999,E2 -10349.999} C_VEL
LIN {X 0,Y 410.012,Z 836.112,A -85,B 0,C 180,E1 -10351.964,E2 -10351.964} C_VEL
LIN {X 0,Y 410.039,Z 835.147,A -85,B 0,C 180,E1 -10352.947,E2 -10352.947} C_VEL
LIN {X 0,Y 410.036,Z 833.786,A -85,B 0,C 180,E1 -10353.93,E2 -10353.93} C_VEL
LIN {X 0,Y 410.258,Z 830.917,A -85,B 0,C 180,E1 -10355.405,E2 -10355.405} C_VEL
LIN {X 0,Y 410.428,Z 827.02,A -85,B 0,C 180,E1 -10356.883,E2 -10356.883} C_VEL
LIN {X 0,Y 410.741,Z 821.975,A -85,B 0,C 180,E1 -10358.362,E2 -10358.362} C_VEL
LIN {X 0,Y 411.221,Z 815.613,A -85,B 0,C 180,E1 -10359.839,E2 -10359.839} C_VEL
LIN {X 0,Y 411.862,Z 807.697,A -85,B 0,C 180,E1 -10361.316,E2 -10361.316} C_VEL
LIN {X 0,Y 412.5,Z 799.606,A -85,B 0,C 180,E1 -10362.545,E2 -10362.545} C_VEL
LIN {X 0,Y 413.322,Z 789.676,A -85,B 0,C 180,E1 -10363.77,E2 -10363.77} C_VEL
LIN {X 0,Y 414.026,Z 778.523,A -85,B 0,C 180,E1 -10364.876,E2 -10364.876} C_VEL
LIN {X 0,Y 414.761,Z 767.593,A -85,B 0,C 180,E1 -10365.73,E2 -10365.73} C_VEL
LIN {X 0,Y 415.376,Z 755.311,A -85,B 0,C 180,E1 -10366.462,E2 -10366.462} C_VEL
LIN {X 0,Y 415.951,Z 741.718,A -85,B 0,C 180,E1 -10367.039,E2 -10367.039} C_VEL
LIN {X 0,Y 416.244,Z 729.014,A -85,B 0,C 180,E1 -10367.375,E2 -10367.375} C_VEL
LIN {X 0,Y 417.215,Z 643.933,A -85,B 0,C 180,E1 -10368.854,E2 -10368.854} C_VEL
LIN {X 0,Y 413.733,Z 623.375,A -85,B 0,C 180,E1 -10369.411,E2 -10369.411} C_VEL
LIN {X 0,Y 414.395,Z 604.823,A -85,B 0,C 180,E1 -10372.431,E2 -10372.431} C_VEL
LIN {X 0,Y 415.328,Z 586.766,A -85,B 0,C 180,E1 -10375.561,E2 -10375.561} C_VEL
LIN {X 0,Y 416.053,Z 571.663,A -85,B 0,C 180,E1 -10378.226,E2 -10378.226} C_VEL
LIN {X 0,Y 414.22,Z 562.08,A -85,B 0,C 180,E1 -10380.082,E2 -10380.082} C_VEL
LIN {X 0,Y 411.202,Z 549.267,A -85,B 0,C 180,E1 -10382.641,E2 -10382.641} C_VEL
LIN {X 0,Y 411.196,Z 549.263,A -85,B 0,C 180,E1 -10385.527,E2 -10385.527} C_VEL
LIN {X 0,Y 411.22,Z 549.256,A -85,B 0,C 180,E1 -10389.222,E2 -10389.222} C_VEL
LIN {X 0,Y 411.179,Z 549.26,A -85,B 0,C 180,E1 -10392.695,E2 -10392.695} C_VEL
LIN {X 0,Y 411.222,Z 549.261,A -85,B 0,C 180,E1 -10395.871,E2 -10395.871} C_VEL
LIN {X 0,Y 411.275,Z 549.41,A -85,B 0,C 180,E1 -10399.561,E2 -10399.561} C_VEL
LIN {X 0,Y 416.427,Z 564.226,A -85,B 0,C 180,E1 -10400.076,E2 -10400.076} C_VEL
LIN {X 0,Y 415.497,Z 629.749,A -85,B 0,C 180,E1 -10401.353,E2 -10401.353} C_VEL
LIN {X 0,Y 415.452,Z 643.524,A -85,B 0,C 180,E1 -10401.831,E2 -10401.831} C_VEL
LIN {X 0,Y 415.181,Z 655.975,A -85,B 0,C 180,E1 -10402.454,E2 -10402.454} C_VEL
LIN {X 0,Y 414.799,Z 667.185,A -85,B 0,C 180,E1 -10403.202,E2 -10403.202} C_VEL
LIN {X 0,Y 414.274,Z 678.716,A -85,B 0,C 180,E1 -10404.179,E2 -10404.179} C_VEL
LIN {X 0,Y 413.731,Z 689.445,A -85,B 0,C 180,E1 -10405.315,E2 -10405.315} C_VEL
LIN {X 0,Y 413.227,Z 698.101,A -85,B 0,C 180,E1 -10406.444,E2 -10406.444} C_VEL
LIN {X 0,Y 412.72,Z 706.904,A -85,B 0,C 180,E1 -10407.85,E2 -10407.85} C_VEL
LIN {X 0,Y 412.275,Z 714.003,A -85,B 0,C 180,E1 -10409.242,E2 -10409.242} C_VEL
LIN {X 0,Y 411.902,Z 719.163,A -85,B 0,C 180,E1 -10410.476,E2 -10410.476} C_VEL
LIN {X 0,Y 411.667,Z 724.283,A -85,B 0,C 180,E1 -10411.999,E2 -10411.999} C_VEL
LIN {X 0,Y 411.428,Z 728.451,A -85,B 0,C 180,E1 -10413.632,E2 -10413.632} C_VEL
LIN {X 0,Y 411.271,Z 730.803,A -85,B 0,C 180,E1 -10414.913,E2 -10414.913} C_VEL
LIN {X 0,Y 411.227,Z 732.007,A -85,B 0,C 180,E1 -10415.784,E2 -10415.784} C_VEL
LIN {X 0,Y 411.221,Z 733.332,A -85,B 0,C 180,E1 -10417.348,E2 -10417.348} C_VEL
LIN {X 0,Y 411.279,Z 733.614,A -85,B 0,C 180,E1 -10418.97,E2 -10418.97} C_VEL
LIN {X 0,Y 411.357,Z 733.174,A -85,B 0,C 180,E1 -10420.019,E2 -10420.019} C_VEL
LIN {X 0,Y 411.479,Z 732.291,A -85,B 0,C 180,E1 -10421.064,E2 -10421.064} C_VEL
LIN {X 0,Y 411.783,Z 729.607,A -85,B 0,C 180,E1 -10422.889,E2 -10422.889} C_VEL
LIN {X 0,Y 412.196,Z 725.428,A -85,B 0,C 180,E1 -10424.676,E2 -10424.676} C_VEL
LIN {X 0,Y 412.663,Z 720.55,A -85,B 0,C 180,E1 -10426.206,E2 -10426.206} C_VEL
LIN {X 0,Y 413.231,Z 714.328,A -85,B 0,C 180,E1 -10427.726,E2 -10427.726} C_VEL
LIN {X 0,Y 413.879,Z 706.449,A -85,B 0,C 180,E1 -10429.234,E2 -10429.234} C_VEL
LIN {X 0,Y 414.51,Z 698.372,A -85,B 0,C 180,E1 -10430.485,E2 -10430.485} C_VEL
LIN {X 0,Y 415.187,Z 688.502,A -85,B 0,C 180,E1 -10431.727,E2 -10431.727} C_VEL
LIN {X 0,Y 415.797,Z 678.686,A -85,B 0,C 180,E1 -10432.717,E2 -10432.717} C_VEL
LIN {X 0,Y 416.349,Z 666.459,A -85,B 0,C 180,E1 -10433.701,E2 -10433.701} C_VEL
LIN {X 0,Y 416.787,Z 654.05,A -85,B 0,C 180,E1 -10434.455,E2 -10434.455} C_VEL
LIN {X 0,Y 416.962,Z 640.276,A -85,B 0,C 180,E1 -10435.054,E2 -10435.054} C_VEL
LIN {X 0,Y 416.972,Z 626.811,A -85,B 0,C 180,E1 -10435.42,E2 -10435.42} C_VEL
LIN {X 0,Y 418.041,Z 565.523,A -85,B 0,C 180,E1 -10436.672,E2 -10436.672} C_VEL
LIN {X 0,Y 411.531,Z 549.528,A -85,B 0,C 180,E1 -10437.431,E2 -10437.431} C_VEL
LIN {X 0,Y 411.476,Z 549.23,A -85,B 0,C 180,E1 -10437.491,E2 -10437.491} C_VEL
LIN {X 0,Y 411.633,Z 549.213,A -85,B 0,C 180,E1 -10440,E2 -10440} C_VEL
LIN {X 0,Y 411.458,Z 549.234,A -85,B 0,C 180,E1 -10442.937,E2 -10442.937} C_VEL
LIN {X 0,Y 411.483,Z 549.227,A -85,B 0,C 180,E1 -10445.882,E2 -10445.882} C_VEL
LIN {X 0,Y 411.471,Z 549.226,A -85,B 0,C 180,E1 -10447.854,E2 -10447.854} C_VEL
LIN {X 0,Y 411.289,Z 549.252,A -85,B 0,C 180,E1 -10451.833,E2 -10451.833} C_VEL
LIN {X 0,Y 411.252,Z 549.256,A -85,B 0,C 180,E1 -10454.853,E2 -10454.853} C_VEL
LIN {X 0,Y 411.242,Z 549.257,A -85,B 0,C 180,E1 -10457.916,E2 -10457.916} C_VEL
LIN {X 0,Y 411.186,Z 549.266,A -85,B 0,C 180,E1 -10461.035,E2 -10461.035} C_VEL
LIN {X 0,Y 411.217,Z 549.261,A -85,B 0,C 180,E1 -10464.216,E2 -10464.216} C_VEL
LIN {X 0,Y 411.25,Z 549.255,A -85,B 0,C 180,E1 -10467.478,E2 -10467.478} C_VEL
LIN {X 0,Y 411.189,Z 549.267,A -85,B 0,C 180,E1 -10470.848,E2 -10470.848} C_VEL
LIN {X 0,Y 411.198,Z 549.262,A -85,B 0,C 180,E1 -10474.334,E2 -10474.334} C_VEL
LIN {X 0,Y 411.198,Z 549.26,A -85,B 0,C 180,E1 -10477.974,E2 -10477.974} C_VEL
LIN {X 0,Y 411.204,Z 549.267,A -85,B 0,C 180,E1 -10481.237,E2 -10481.237} C_VEL
LIN {X 0,Y 411.228,Z 549.264,A -85,B 0,C 180,E1 -10484.483,E2 -10484.483} C_VEL
LIN {X 0,Y 411.227,Z 549.261,A -85,B 0,C 180,E1 -10487.298,E2 -10487.298} C_VEL
LIN {X 0,Y 411.227,Z 549.262,A -85,B 0,C 180,E1 -10490.779,E2 -10490.779} C_VEL
LIN {X 0,Y 411.196,Z 549.27,A -85,B 0,C 180,E1 -10494.473,E2 -10494.473} C_VEL
LIN {X 0,Y 411.214,Z 549.277,A -85,B 0,C 180,E1 -10496.737,E2 -10496.737} C_VEL
LIN {X 0,Y 414.559,Z 562.698,A -85,B 0,C 180,E1 -10499.432,E2 -10499.432} C_VEL
LIN {X 0,Y 416.413,Z 571.686,A -85,B 0,C 180,E1 -10501.099,E2 -10501.099} C_VEL
LIN {X 0,Y 416.337,Z 575.837,A -85,B 0,C 180,E1 -10501.795,E2 -10501.795} C_VEL
LIN {X 0,Y 414.775,Z 595.556,A -85,B 0,C 180,E1 -10504.939,E2 -10504.939} C_VEL
LIN {X 0,Y 413.25,Z 618.823,A -85,B 0,C 180,E1 -10508.554,E2 -10508.554} C_VEL
LIN {X 0,Y 412.703,Z 629.683,A -85,B 0,C 180,E1 -10510.214,E2 -10510.214} C_VEL
LIN {X 0,Y 415.787,Z 657.157,A -85,B 0,C 180,E1 -10510.981,E2 -10510.981} C_VEL
LIN {X 0,Y 416.883,Z 671.56,A -85,B 0,C 180,E1 -10511.337,E2 -10511.337} C_VEL
LIN {X 0,Y 415.432,Z 758.313,A -85,B 0,C 180,E1 -10513.034,E2 -10513.034} C_VEL
LIN {X 0,Y 414.93,Z 771.685,A -85,B 0,C 180,E1 -10513.488,E2 -10513.488} C_VEL
LIN {X 0,Y 414.338,Z 784.268,A -85,B 0,C 180,E1 -10514.128,E2 -10514.128} C_VEL
LIN {X 0,Y 413.626,Z 796.629,A -85,B 0,C 180,E1 -10514.983,E2 -10514.983} C_VEL
LIN {X 0,Y 412.894,Z 807.805,A -85,B 0,C 180,E1 -10515.982,E2 -10515.982} C_VEL
LIN {X 0,Y 412.134,Z 818.479,A -85,B 0,C 180,E1 -10517.193,E2 -10517.193} C_VEL
LIN {X 0,Y 411.491,Z 827.282,A -85,B 0,C 180,E1 -10518.424,E2 -10518.424} C_VEL
LIN {X 0,Y 411.024,Z 834.531,A -85,B 0,C 180,E1 -10519.658,E2 -10519.658} C_VEL
LIN {X 0,Y 410.591,Z 841.632,A -85,B 0,C 180,E1 -10521.139,E2 -10521.139} C_VEL
LIN {X 0,Y 410.289,Z 847.27,A -85,B 0,C 180,E1 -10522.62,E2 -10522.62} C_VEL
LIN {X 0,Y 410.112,Z 851.69,A -85,B 0,C 180,E1 -10524.099,E2 -10524.099} C_VEL
LIN {X 0,Y 410.143,Z 854.02,A -85,B 0,C 180,E1 -10525.086,E2 -10525.086} C_VEL
LIN {X 0,Y 410.029,Z 855.914,A -85,B 0,C 180,E1 -10526.07,E2 -10526.07} C_VEL
LIN {X 0,Y 410.036,Z 857.345,A -85,B 0,C 180,E1 -10527.053,E2 -10527.053} C_VEL
LIN {X 0,Y 410.065,Z 858.354,A -85,B 0,C 180,E1 -10528.037,E2 -10528.037} C_VEL
LIN {X 0,Y 410.041,Z 858.969,A -85,B 0,C 180,E1 -10529.019,E2 -10529.019} C_VEL
LIN {X 0,Y 410.046,Z 859.19,A -85,B 0,C 180,E1 -10530.001,E2 -10530.001} C_VEL
LIN {X 0,Y 410.06,Z 858.349,A -85,B 0,C 180,E1 -10531.965,E2 -10531.965} C_VEL
LIN {X 0,Y 410.024,Z 857.337,A -85,B 0,C 180,E1 -10532.948,E2 -10532.948} C_VEL
LIN {X 0,Y 410.015,Z 855.902,A -85,B 0,C 180,E1 -10533.932,E2 -10533.932} C_VEL
LIN {X 0,Y 410.128,Z 852.92,A -85,B 0,C 180,E1 -10535.409,E2 -10535.409} C_VEL
LIN {X 0,Y 410.252,Z 848.87,A -85,B 0,C 180,E1 -10536.888,E2 -10536.888} C_VEL
LIN {X 0,Y 410.493,Z 842.614,A -85,B 0,C 180,E1 -10538.616,E2 -10538.616} C_VEL
LIN {X 0,Y 410.895,Z 835.789,A -85,B 0,C 180,E1 -10540.098,E2 -10540.098} C_VEL
LIN {X 0,Y 411.33,Z 828.813,A -85,B 0,C 180,E1 -10541.332,E2 -10541.332} C_VEL
LIN {X 0,Y 411.979,Z 820.382,A -85,B 0,C 180,E1 -10542.563,E2 -10542.563} C_VEL
LIN {X 0,Y 412.681,Z 809.923,A -85,B 0,C 180,E1 -10543.794,E2 -10543.794} C_VEL
LIN {X 0,Y 413.375,Z 799.549,A -85,B 0,C 180,E1 -10544.776,E2 -10544.776} C_VEL
LIN {X 0,Y 414.099,Z 788.112,A -85,B 0,C 180,E1 -10545.631,E2 -10545.631} C_VEL
LIN {X 0,Y 414.73,Z 776.217,A -85,B 0,C 180,E1 -10546.301,E2 -10546.301} C_VEL
LIN {X 0,Y 415.25,Z 763.342,A -85,B 0,C 180,E1 -10546.817,E2 -10546.817} C_VEL
LIN {X 0,Y 415.539,Z 751.218,A -85,B 0,C 180,E1 -10547.122,E2 -10547.122} C_VEL
LIN {X 0,Y 416.403,Z 671.052,A -85,B 0,C 180,E1 -10548.5,E2 -10548.5} C_VEL
LIN {X 0,Y 412.394,Z 636.734,A -85,B 0,C 180,E1 -10549.324,E2 -10549.324} C_VEL
LIN {X 0,Y 412.325,Z 635.119,A -85,B 0,C 180,E1 -10549.413,E2 -10549.413} C_VEL
LIN {X 0,Y 413.481,Z 613.773,A -85,B 0,C 180,E1 -10553.013,E2 -10553.013} C_VEL
LIN {X 0,Y 414.869,Z 592.35,A -85,B 0,C 180,E1 -10556.675,E2 -10556.675} C_VEL
LIN {X 0,Y 416.197,Z 573.831,A -85,B 0,C 180,E1 -10559.878,E2 -10559.878} C_VEL
LIN {X 0,Y 415.669,Z 569.053,A -85,B 0,C 180,E1 -10560.761,E2 -10560.761} C_VEL
LIN {X 0,Y 411.959,Z 552.403,A -85,B 0,C 180,E1 -10564.024,E2 -10564.024} C_VEL
LIN {X 0,Y 411.232,Z 549.262,A -85,B 0,C 180,E1 -10564.677,E2 -10564.677} C_VEL
LIN {X 0,Y 411.208,Z 549.262,A -85,B 0,C 180,E1 -10568.169,E2 -10568.169} C_VEL
LIN {X 0,Y 411.166,Z 549.271,A -85,B 0,C 180,E1 -10571.228,E2 -10571.228} C_VEL
LIN {X 0,Y 411.179,Z 549.257,A -85,B 0,C 180,E1 -10574.49,E2 -10574.49} C_VEL
LIN {X 0,Y 411.181,Z 549.256,A -85,B 0,C 180,E1 -10578.195,E2 -10578.195} C_VEL
LIN {X 0,Y 411.22,Z 549.261,A -85,B 0,C 180,E1 -10580.776,E2 -10580.776} C_VEL
LIN {X 0,Y 411.201,Z 549.256,A -85,B 0,C 180,E1 -10584.471,E2 -10584.471} C_VEL
LIN {X 0,Y 411.208,Z 549.263,A -85,B 0,C 180,E1 -10586.873,E2 -10586.873} C_VEL
LIN {X 0,Y 411.234,Z 549.253,A -85,B 0,C 180,E1 -10590.644,E2 -10590.644} C_VEL
LIN {X 0,Y 411.239,Z 549.253,A -85,B 0,C 180,E1 -10593.619,E2 -10593.619} C_VEL
LIN {X 0,Y 411.197,Z 549.256,A -85,B 0,C 180,E1 -10596.852,E2 -10596.852} C_VEL
LIN {X 0,Y 411.215,Z 549.256,A -85,B 0,C 180,E1 -10600.051,E2 -10600.051} C_VEL
LIN {X 0,Y 411.264,Z 549.242,A -85,B 0,C 180,E1 -10603.131,E2 -10603.131} C_VEL
LIN {X 0,Y 411.306,Z 549.248,A -85,B 0,C 180,E1 -10606.896,E2 -10606.896} C_VEL
LIN {X 0,Y 411.293,Z 549.24,A -85,B 0,C 180,E1 -10610.161,E2 -10610.161} C_VEL
LIN {X 0,Y 411.456,Z 549.23,A -85,B 0,C 180,E1 -10613.133,E2 -10613.133} C_VEL
LIN {X 0,Y 411.311,Z 549.247,A -85,B 0,C 180,E1 -10615.099,E2 -10615.099} C_VEL
LIN {X 0,Y 411.511,Z 549.213,A -85,B 0,C 180,E1 -10618.043,E2 -10618.043} C_VEL
LIN {X 0,Y 411.64,Z 549.21,A -85,B 0,C 180,E1 -10620,E2 -10620} C_VEL
LIN {X 0,Y 411.459,Z 549.226,A -85,B 0,C 180,E1 -10622.937,E2 -10622.937} C_VEL
LIN {X 0,Y 411.45,Z 549.222,A -85,B 0,C 180,E1 -10626.642,E2 -10626.642} C_VEL
LIN {X 0,Y 411.305,Z 549.25,A -85,B 0,C 180,E1 -10629.839,E2 -10629.839} C_VEL
LIN {X 0,Y 411.306,Z 549.235,A -85,B 0,C 180,E1 -10633.104,E2 -10633.104} C_VEL
LIN {X 0,Y 411.258,Z 549.253,A -85,B 0,C 180,E1 -10636.889,E2 -10636.889} C_VEL
LIN {X 0,Y 411.231,Z 549.25,A -85,B 0,C 180,E1 -10639.987,E2 -10639.987} C_VEL
LIN {X 0,Y 411.204,Z 549.26,A -85,B 0,C 180,E1 -10643.148,E2 -10643.148} C_VEL
LIN {X 0,Y 411.239,Z 549.255,A -85,B 0,C 180,E1 -10646.381,E2 -10646.381} C_VEL
LIN {X 0,Y 411.202,Z 549.263,A -85,B 0,C 180,E1 -10649.713,E2 -10649.713} C_VEL
LIN {X 0,Y 411.208,Z 549.262,A -85,B 0,C 180,E1 -10653.156,E2 -10653.156} C_VEL
LIN {X 0,Y 411.194,Z 549.267,A -85,B 0,C 180,E1 -10656.553,E2 -10656.553} C_VEL
LIN {X 0,Y 411.214,Z 549.259,A -85,B 0,C 180,E1 -10659.728,E2 -10659.728} C_VEL
LIN {X 0,Y 411.175,Z 549.26,A -85,B 0,C 180,E1 -10663.134,E2 -10663.134} C_VEL
LIN {X 0,Y 411.169,Z 549.266,A -85,B 0,C 180,E1 -10665.881,E2 -10665.881} C_VEL
LIN {X 0,Y 411.164,Z 549.265,A -85,B 0,C 180,E1 -10668.772,E2 -10668.772} C_VEL
LIN {X 0,Y 411.21,Z 549.254,A -85,B 0,C 180,E1 -10671.831,E2 -10671.831} C_VEL
LIN {X 0,Y 411.214,Z 549.263,A -85,B 0,C 180,E1 -10675.121,E2 -10675.121} C_VEL
LIN {X 0,Y 411.169,Z 549.267,A -85,B 0,C 180,E1 -10678.003,E2 -10678.003} C_VEL
LIN {X 0,Y 411.248,Z 549.463,A -85,B 0,C 180,E1 -10679.048,E2 -10679.048} C_VEL
LIN {X 0,Y 414.947,Z 564.677,A -85,B 0,C 180,E1 -10681.731,E2 -10681.731} C_VEL
LIN {X 0,Y 416.468,Z 572.41,A -85,B 0,C 180,E1 -10683.074,E2 -10683.074} C_VEL
LIN {X 0,Y 415.631,Z 587.965,A -85,B 0,C 180,E1 -10685.526,E2 -10685.526} C_VEL
LIN {X 0,Y 414.506,Z 611.74,A -85,B 0,C 180,E1 -10689.141,E2 -10689.141} C_VEL
LIN {X 0,Y 414.135,Z 622.553,A -85,B 0,C 180,E1 -10690.695,E2 -10690.695} C_VEL
LIN {X 0,Y 417.208,Z 642.188,A -85,B 0,C 180,E1 -10691.21,E2 -10691.21} C_VEL
LIN {X 0,Y 416.178,Z 733.074,A -85,B 0,C 180,E1 -10692.811,E2 -10692.811} C_VEL
LIN {X 0,Y 415.745,Z 746.637,A -85,B 0,C 180,E1 -10693.235,E2 -10693.235} C_VEL
LIN {X 0,Y 415.106,Z 759.235,A -85,B 0,C 180,E1 -10693.841,E2 -10693.841} C_VEL
LIN {X 0,Y 414.441,Z 771.363,A -85,B 0,C 180,E1 -10694.635,E2 -10694.635} C_VEL
LIN {X 0,Y 413.756,Z 782.64,A -85,B 0,C 180,E1 -10695.595,E2 -10695.595} C_VEL
LIN {X 0,Y 413.024,Z 793.112,A -85,B 0,C 180,E1 -10696.719,E2 -10696.719} C_VEL
LIN {X 0,Y 412.272,Z 802.404,A -85,B 0,C 180,E1 -10697.946,E2 -10697.946} C_VEL
LIN {X 0,Y 411.662,Z 810.022,A -85,B 0,C 180,E1 -10699.175,E2 -10699.175} C_VEL
LIN {X 0,Y 411.435,Z 812.821,A -85,B 0,C 180,E1 -10699.697,E2 -10699.697} C_VEL
LIN {X 0,Y 410.49,Z 816.217,A -85,B 0,C 180,E1 -10700.36,E2 -10700.36} C_VEL
LIN {X 0,Y 407.278,Z 821.337,A -85,B 0,C 180,E1 -10701.463,E2 -10701.463} C_VEL
LIN {X 0,Y 404.148,Z 825.774,A -85,B 0,C 180,E1 -10702.635,E2 -10702.635} C_VEL
LIN {X 0,Y 403.346,Z 828.065,A -85,B 0,C 180,E1 -10703.4,E2 -10703.4} C_VEL
LIN {X 0,Y 403.101,Z 831.951,A -85,B 0,C 180,E1 -10704.998,E2 -10704.998} C_VEL
LIN {X 0,Y 402.956,Z 833.812,A -85,B 0,C 180,E1 -10705.999,E2 -10705.999} C_VEL
LIN {X 0,Y 402.955,Z 835.232,A -85,B 0,C 180,E1 -10707,E2 -10707} C_VEL
LIN {X 0,Y 402.926,Z 836.228,A -85,B 0,C 180,E1 -10708,E2 -10708} C_VEL
LIN {X 0,Y 402.851,Z 837.081,A -85,B 0,C 180,E1 -10709.999,E2 -10709.999} C_VEL
LIN {X 0,Y 402.867,Z 836.89,A -85,B 0,C 180,E1 -10710.999,E2 -10710.999} C_VEL
LIN {X 0,Y 402.925,Z 836.304,A -85,B 0,C 180,E1 -10711.998,E2 -10711.998} C_VEL
LIN {X 0,Y 402.941,Z 835.34,A -85,B 0,C 180,E1 -10712.999,E2 -10712.999} C_VEL
LIN {X 0,Y 402.954,Z 833.978,A -85,B 0,C 180,E1 -10714,E2 -10714} C_VEL
LIN {X 0,Y 403.184,Z 831.108,A -85,B 0,C 180,E1 -10715.501,E2 -10715.501} C_VEL
LIN {X 0,Y 403.363,Z 827.211,A -85,B 0,C 180,E1 -10717.005,E2 -10717.005} C_VEL
LIN {X 0,Y 403.695,Z 822.164,A -85,B 0,C 180,E1 -10718.509,E2 -10718.509} C_VEL
LIN {X 0,Y 404.204,Z 815.801,A -85,B 0,C 180,E1 -10720.012,E2 -10720.012} C_VEL
LIN {X 0,Y 404.869,Z 807.883,A -85,B 0,C 180,E1 -10721.514,E2 -10721.514} C_VEL
LIN {X 0,Y 405.579,Z 799.788,A -85,B 0,C 180,E1 -10722.763,E2 -10722.763} C_VEL
LIN {X 0,Y 406.415,Z 789.854,A -85,B 0,C 180,E1 -10724.009,E2 -10724.009} C_VEL
LIN {X 0,Y 407.17,Z 778.695,A -85,B 0,C 180,E1 -10725.132,E2 -10725.132} C_VEL
LIN {X 0,Y 407.93,Z 767.758,A -85,B 0,C 180,E1 -10726,E2 -10726} C_VEL
LIN {X 0,Y 408.586,Z 755.461,A -85,B 0,C 180,E1 -10726.744,E2 -10726.744} C_VEL
LIN {X 0,Y 409.132,Z 742.679,A -85,B 0,C 180,E1 -10727.3,E2 -10727.3} C_VEL
LIN {X 0,Y 409.452,Z 730.634,A -85,B 0,C 180,E1 -10727.64,E2 -10727.64} C_VEL
LIN {X 0,Y 410.48,Z 644.663,A -85,B 0,C 180,E1 -10729.162,E2 -10729.162} C_VEL
LIN {X 0,Y 406.893,Z 623.516,A -85,B 0,C 180,E1 -10729.752,E2 -10729.752} C_VEL
LIN {X 0,Y 407.586,Z 604.782,A -85,B 0,C 180,E1 -10732.827,E2 -10732.827} C_VEL
LIN {X 0,Y 408.591,Z 586.547,A -85,B 0,C 180,E1 -10736.014,E2 -10736.014} C_VEL
LIN {X 0,Y 409.235,Z 573.371,A -85,B 0,C 180,E1 -10738.375,E2 -10738.375} C_VEL
LIN {X 0,Y 407.685,Z 565.061,A -85,B 0,C 180,E1 -10739.994,E2 -10739.994} C_VEL
LIN {X 0,Y 404.629,Z 552.091,A -85,B 0,C 180,E1 -10742.576,E2 -10742.576} C_VEL
LIN {X 0,Y 404.164,Z 550.14,A -85,B 0,C 180,E1 -10742.985,E2 -10742.985} C_VEL
LIN {X 0,Y 404.141,Z 550.14,A -85,B 0,C 180,E1 -10746.245,E2 -10746.245} C_VEL
LIN {X 0,Y 404.155,Z 550.139,A -85,B 0,C 180,E1 -10748.755,E2 -10748.755} C_VEL
LIN {X 0,Y 404.12,Z 550.146,A -85,B 0,C 180,E1 -10751.599,E2 -10751.599} C_VEL
LIN {X 0,Y 404.151,Z 550.133,A -85,B 0,C 180,E1 -10754.523,E2 -10754.523} C_VEL
LIN {X 0,Y 404.201,Z 550.139,A -85,B 0,C 180,E1 -10757.304,E2 -10757.304} C_VEL
LIN {X 0,Y 404.193,Z 550.14,A -85,B 0,C 180,E1 -10759.269,E2 -10759.269} C_VEL
LIN {X 0,Y 409.519,Z 565.49,A -85,B 0,C 180,E1 -10759.82,E2 -10759.82} C_VEL
LIN {X 0,Y 408.647,Z 631.14,A -85,B 0,C 180,E1 -10761.136,E2 -10761.136} C_VEL
LIN {X 0,Y 408.579,Z 645.192,A -85,B 0,C 180,E1 -10761.641,E2 -10761.641} C_VEL
LIN {X 0,Y 408.278,Z 657.106,A -85,B 0,C 180,E1 -10762.255,E2 -10762.255} C_VEL
LIN {X 0,Y 407.854,Z 668.86,A -85,B 0,C 180,E1 -10763.061,E2 -10763.061} C_VEL
LIN {X 0,Y 407.341,Z 680.546,A -85,B 0,C 180,E1 -10764.083,E2 -10764.083} C_VEL
LIN {X 0,Y 406.765,Z 691.083,A -85,B 0,C 180,E1 -10765.238,E2 -10765.238} C_VEL
LIN {X 0,Y 406.116,Z 701.54,A -85,B 0,C 180,E1 -10766.671,E2 -10766.671} C_VEL
LIN {X 0,Y 405.628,Z 709.899,A -85,B 0,C 180,E1 -10768.098,E2 -10768.098} C_VEL
LIN {X 0,Y 405.096,Z 717.779,A -85,B 0,C 180,E1 -10769.793,E2 -10769.793} C_VEL
LIN {X 0,Y 404.702,Z 723.873,A -85,B 0,C 180,E1 -10771.474,E2 -10771.474} C_VEL
LIN {X 0,Y 404.469,Z 728.404,A -85,B 0,C 180,E1 -10773.142,E2 -10773.142} C_VEL
LIN {X 0,Y 404.268,Z 731.459,A -85,B 0,C 180,E1 -10774.684,E2 -10774.684} C_VEL
LIN {X 0,Y 404.163,Z 733.672,A -85,B 0,C 180,E1 -10776.425,E2 -10776.425} C_VEL
LIN {X 0,Y 404.2,Z 734.433,A -85,B 0,C 180,E1 -10777.51,E2 -10777.51} C_VEL
LIN {X 0,Y 404.228,Z 734.667,A -85,B 0,C 180,E1 -10778.585,E2 -10778.585} C_VEL
LIN {X 0,Y 404.321,Z 734.402,A -85,B 0,C 180,E1 -10779.819,E2 -10779.819} C_VEL
LIN {X 0,Y 404.422,Z 733.783,A -85,B 0,C 180,E1 -10780.72,E2 -10780.72} C_VEL
LIN {X 0,Y 404.583,Z 732.61,A -85,B 0,C 180,E1 -10781.779,E2 -10781.779} C_VEL
LIN {X 0,Y 404.908,Z 729.985,A -85,B 0,C 180,E1 -10783.358,E2 -10783.358} C_VEL
LIN {X 0,Y 405.301,Z 726.246,A -85,B 0,C 180,E1 -10784.924,E2 -10784.924} C_VEL
LIN {X 0,Y 405.823,Z 721.248,A -85,B 0,C 180,E1 -10786.492,E2 -10786.492} C_VEL
LIN {X 0,Y 406.417,Z 714.957,A -85,B 0,C 180,E1 -10788.023,E2 -10788.023} C_VEL
LIN {X 0,Y 407.066,Z 707.428,A -85,B 0,C 180,E1 -10789.479,E2 -10789.479} C_VEL
LIN {X 0,Y 407.794,Z 698.811,A -85,B 0,C 180,E1 -10790.827,E2 -10790.827} C_VEL
LIN {X 0,Y 408.489,Z 688.79,A -85,B 0,C 180,E1 -10792.089,E2 -10792.089} C_VEL
LIN {X 0,Y 409.205,Z 677.457,A -85,B 0,C 180,E1 -10793.219,E2 -10793.219} C_VEL
LIN {X 0,Y 409.787,Z 666.309,A -85,B 0,C 180,E1 -10794.094,E2 -10794.094} C_VEL
LIN {X 0,Y 410.162,Z 654.312,A -85,B 0,C 180,E1 -10794.814,E2 -10794.814} C_VEL
LIN {X 0,Y 410.363,Z 640.99,A -85,B 0,C 180,E1 -10795.395,E2 -10795.395} C_VEL
LIN {X 0,Y 410.353,Z 627.719,A -85,B 0,C 180,E1 -10795.758,E2 -10795.758} C_VEL
LIN {X 0,Y 411.458,Z 567.288,A -85,B 0,C 180,E1 -10797.026,E2 -10797.026} C_VEL
LIN {X 0,Y 404.516,Z 550.427,A -85,B 0,C 180,E1 -10797.869,E2 -10797.869} C_VEL
LIN {X 0,Y 404.451,Z 550.106,A -85,B 0,C 180,E1 -10797.896,E2 -10797.896} C_VEL
LIN {X 0,Y 404.602,Z 550.089,A -85,B 0,C 180,E1 -10800,E2 -10800} C_VEL
LIN {X 0,Y 404.415,Z 550.11,A -85,B 0,C 180,E1 -10802.988,E2 -10802.988} C_VEL
LIN {X 0,Y 404.429,Z 550.106,A -85,B 0,C 180,E1 -10805.985,E2 -10805.985} C_VEL
LIN {X 0,Y 404.412,Z 550.105,A -85,B 0,C 180,E1 -10807.992,E2 -10807.992} C_VEL
LIN {X 0,Y 404.26,Z 550.128,A -85,B 0,C 180,E1 -10812.041,E2 -10812.041} C_VEL
LIN {X 0,Y 404.197,Z 550.132,A -85,B 0,C 180,E1 -10815.118,E2 -10815.118} C_VEL
LIN {X 0,Y 404.2,Z 550.136,A -85,B 0,C 180,E1 -10818.239,E2 -10818.239} C_VEL
LIN {X 0,Y 404.129,Z 550.144,A -85,B 0,C 180,E1 -10821.42,E2 -10821.42} C_VEL
LIN {X 0,Y 404.168,Z 550.141,A -85,B 0,C 180,E1 -10824.666,E2 -10824.666} C_VEL
LIN {X 0,Y 404.189,Z 550.134,A -85,B 0,C 180,E1 -10828,E2 -10828} C_VEL
LIN {X 0,Y 404.134,Z 550.143,A -85,B 0,C 180,E1 -10831.56,E2 -10831.56} C_VEL
LIN {X 0,Y 404.177,Z 550.136,A -85,B 0,C 180,E1 -10835.017,E2 -10835.017} C_VEL
LIN {X 0,Y 404.157,Z 550.144,A -85,B 0,C 180,E1 -10838.757,E2 -10838.757} C_VEL
LIN {X 0,Y 404.185,Z 550.139,A -85,B 0,C 180,E1 -10841.612,E2 -10841.612} C_VEL
LIN {X 0,Y 404.192,Z 550.14,A -85,B 0,C 180,E1 -10844.531,E2 -10844.531} C_VEL
LIN {X 0,Y 404.205,Z 550.135,A -85,B 0,C 180,E1 -10847.307,E2 -10847.307} C_VEL
LIN {X 0,Y 404.164,Z 550.141,A -85,B 0,C 180,E1 -10849.957,E2 -10849.957} C_VEL
LIN {X 0,Y 404.137,Z 550.148,A -85,B 0,C 180,E1 -10853.125,E2 -10853.125} C_VEL
LIN {X 0,Y 404.194,Z 550.195,A -85,B 0,C 180,E1 -10856.284,E2 -10856.284} C_VEL
LIN {X 0,Y 407.563,Z 563.479,A -85,B 0,C 180,E1 -10859.046,E2 -10859.046} C_VEL
LIN {X 0,Y 409.679,Z 573.877,A -85,B 0,C 180,E1 -10861.034,E2 -10861.034} C_VEL
LIN {X 0,Y 408.823,Z 585.117,A -85,B 0,C 180,E1 -10862.901,E2 -10862.901} C_VEL
LIN {X 0,Y 407.123,Z 606.385,A -85,B 0,C 180,E1 -10866.321,E2 -10866.321} C_VEL
LIN {X 0,Y 405.784,Z 628.554,A -85,B 0,C 180,E1 -10869.796,E2 -10869.796} C_VEL
LIN {X 0,Y 408.722,Z 652.762,A -85,B 0,C 180,E1 -10870.502,E2 -10870.502} C_VEL
LIN {X 0,Y 410.238,Z 672.235,A -85,B 0,C 180,E1 -10871.005,E2 -10871.005} C_VEL
LIN {X 0,Y 408.623,Z 759.318,A -85,B 0,C 180,E1 -10872.775,E2 -10872.775} C_VEL
LIN {X 0,Y 408.101,Z 772.29,A -85,B 0,C 180,E1 -10873.236,E2 -10873.236} C_VEL
LIN {X 0,Y 407.505,Z 784.105,A -85,B 0,C 180,E1 -10873.854,E2 -10873.854} C_VEL
LIN {X 0,Y 406.753,Z 796.457,A -85,B 0,C 180,E1 -10874.724,E2 -10874.724} C_VEL
LIN {X 0,Y 405.984,Z 807.457,A -85,B 0,C 180,E1 -10875.72,E2 -10875.72} C_VEL
LIN {X 0,Y 405.173,Z 818.296,A -85,B 0,C 180,E1 -10876.969,E2 -10876.969} C_VEL
LIN {X 0,Y 404.521,Z 827.097,A -85,B 0,C 180,E1 -10878.222,E2 -10878.222} C_VEL
LIN {X 0,Y 403.981,Z 834.343,A -85,B 0,C 180,E1 -10879.476,E2 -10879.476} C_VEL
LIN {X 0,Y 403.552,Z 841.443,A -85,B 0,C 180,E1 -10880.983,E2 -10880.983} C_VEL
LIN {X 0,Y 403.209,Z 847.079,A -85,B 0,C 180,E1 -10882.489,E2 -10882.489} C_VEL
LIN {X 0,Y 403.017,Z 851.498,A -85,B 0,C 180,E1 -10883.995,E2 -10883.995} C_VEL
LIN {X 0,Y 403.049,Z 853.828,A -85,B 0,C 180,E1 -10884.999,E2 -10884.999} C_VEL
LIN {X 0,Y 402.947,Z 855.722,A -85,B 0,C 180,E1 -10886,E2 -10886} C_VEL
LIN {X 0,Y 402.934,Z 857.152,A -85,B 0,C 180,E1 -10887.001,E2 -10887.001} C_VEL
LIN {X 0,Y 402.992,Z 858.162,A -85,B 0,C 180,E1 -10888.002,E2 -10888.002} C_VEL
LIN {X 0,Y 402.962,Z 858.777,A -85,B 0,C 180,E1 -10889.002,E2 -10889.002} C_VEL
LIN {X 0,Y 402.964,Z 858.997,A -85,B 0,C 180,E1 -10890.001,E2 -10890.001} C_VEL
LIN {X 0,Y 402.987,Z 858.156,A -85,B 0,C 180,E1 -10892,E2 -10892} C_VEL
LIN {X 0,Y 402.922,Z 857.144,A -85,B 0,C 180,E1 -10893,E2 -10893} C_VEL
LIN {X 0,Y 402.933,Z 855.709,A -85,B 0,C 180,E1 -10894.001,E2 -10894.001} C_VEL
LIN {X 0,Y 403.025,Z 852.727,A -85,B 0,C 180,E1 -10895.504,E2 -10895.504} C_VEL
LIN {X 0,Y 403.186,Z 848.677,A -85,B 0,C 180,E1 -10897.009,E2 -10897.009} C_VEL
LIN {X 0,Y 403.431,Z 842.421,A -85,B 0,C 180,E1 -10898.768,E2 -10898.768} C_VEL
LIN {X 0,Y 403.881,Z 835.598,A -85,B 0,C 180,E1 -10900.275,E2 -10900.275} C_VEL
LIN {X 0,Y 404.341,Z 828.622,A -85,B 0,C 180,E1 -10901.531,E2 -10901.531} C_VEL
LIN {X 0,Y 405.023,Z 820.194,A -85,B 0,C 180,E1 -10902.782,E2 -10902.782} C_VEL
LIN {X 0,Y 405.783,Z 809.189,A -85,B 0,C 180,E1 -10904.093,E2 -10904.093} C_VEL
LIN {X 0,Y 406.623,Z 797.933,A -85,B 0,C 180,E1 -10905.155,E2 -10905.155} C_VEL
LIN {X 0,Y 407.376,Z 785.969,A -85,B 0,C 180,E1 -10906.024,E2 -10906.024} C_VEL
LIN {X 0,Y 407.976,Z 773.48,A -85,B 0,C 180,E1 -10906.707,E2 -10906.707} C_VEL
LIN {X 0,Y 408.554,Z 761.289,A -85,B 0,C 180,E1 -10907.166,E2 -10907.166} C_VEL
LIN {X 0,Y 408.953,Z 745.809,A -85,B 0,C 180,E1 -10907.503,E2 -10907.503} C_VEL
LIN {X 0,Y 409.687,Z 671.879,A -85,B 0,C 180,E1 -10908.798,E2 -10908.798} C_VEL
LIN {X 0,Y 405.618,Z 636.515,A -85,B 0,C 180,E1 -10909.666,E2 -10909.666} C_VEL
LIN {X 0,Y 405.322,Z 633.631,A -85,B 0,C 180,E1 -10909.829,E2 -10909.829} C_VEL
LIN {X 0,Y 406.484,Z 614.226,A -85,B 0,C 180,E1 -10913.163,E2 -10913.163} C_VEL
LIN {X 0,Y 407.925,Z 592.781,A -85,B 0,C 180,E1 -10916.889,E2 -10916.889} C_VEL
LIN {X 0,Y 409.223,Z 575.837,A -85,B 0,C 180,E1 -10919.871,E2 -10919.871} C_VEL
LIN {X 0,Y 408.862,Z 571.15,A -85,B 0,C 180,E1 -10920.744,E2 -10920.744} C_VEL
LIN {X 0,Y 405.241,Z 554.717,A -85,B 0,C 180,E1 -10924.007,E2 -10924.007} C_VEL
LIN {X 0,Y 404.19,Z 550.14,A -85,B 0,C 180,E1 -10924.978,E2 -10924.978} C_VEL
LIN {X 0,Y 404.158,Z 550.144,A -85,B 0,C 180,E1 -10928.757,E2 -10928.757} C_VEL
LIN {X 0,Y 404.125,Z 550.145,A -85,B 0,C 180,E1 -10931.6,E2 -10931.6} C_VEL
LIN {X 0,Y 404.149,Z 550.133,A -85,B 0,C 180,E1 -10934.522,E2 -10934.522} C_VEL
LIN {X 0,Y 404.142,Z 550.139,A -85,B 0,C 180,E1 -10937.296,E2 -10937.296} C_VEL
LIN {X 0,Y 404.17,Z 550.137,A -85,B 0,C 180,E1 -10939.955,E2 -10939.955} C_VEL
LIN {X 0,Y 404.141,Z 550.135,A -85,B 0,C 180,E1 -10943.124,E2 -10943.124} C_VEL
LIN {X 0,Y 404.146,Z 550.14,A -85,B 0,C 180,E1 -10946.188,E2 -10946.188} C_VEL
LIN {X 0,Y 404.146,Z 550.135,A -85,B 0,C 180,E1 -10949.715,E2 -10949.715} C_VEL
LIN {X 0,Y 404.197,Z 550.137,A -85,B 0,C 180,E1 -10953.123,E2 -10953.123} C_VEL
LIN {X 0,Y 404.175,Z 550.127,A -85,B 0,C 180,E1 -10955.334,E2 -10955.334} C_VEL
LIN {X 0,Y 404.139,Z 550.141,A -85,B 0,C 180,E1 -10958.581,E2 -10958.581} C_VEL
LIN {X 0,Y 404.211,Z 550.118,A -85,B 0,C 180,E1 -10961.762,E2 -10961.762} C_VEL
LIN {X 0,Y 404.207,Z 550.131,A -85,B 0,C 180,E1 -10964.882,E2 -10964.882} C_VEL
LIN {X 0,Y 404.256,Z 550.119,A -85,B 0,C 180,E1 -10967.959,E2 -10967.959} C_VEL
LIN {X 0,Y 404.406,Z 550.108,A -85,B 0,C 180,E1 -10972.129,E2 -10972.129} C_VEL
LIN {X 0,Y 404.423,Z 550.106,A -85,B 0,C 180,E1 -10974.015,E2 -10974.015} C_VEL
LIN {X 0,Y 404.48,Z 550.088,A -85,B 0,C 180,E1 -10978.009,E2 -10978.009} C_VEL
LIN {X 0,Y 404.609,Z 550.085,A -85,B 0,C 180,E1 -10980,E2 -10980} C_VEL
LIN {X 0,Y 404.417,Z 550.104,A -85,B 0,C 180,E1 -10982.988,E2 -10982.988} C_VEL
LIN {X 0,Y 404.396,Z 550.1,A -85,B 0,C 180,E1 -10986.642,E2 -10986.642} C_VEL
LIN {X 0,Y 404.295,Z 550.121,A -85,B 0,C 180,E1 -10989.001,E2 -10989.001} C_VEL
LIN {X 0,Y 404.257,Z 550.114,A -85,B 0,C 180,E1 -10992.042,E2 -10992.042} C_VEL
LIN {X 0,Y 404.207,Z 550.131,A -85,B 0,C 180,E1 -10995.118,E2 -10995.118} C_VEL
LIN {X 0,Y 404.211,Z 550.123,A -85,B 0,C 180,E1 -10998.238,E2 -10998.238} C_VEL
LIN {X 0,Y 404.139,Z 550.139,A -85,B 0,C 180,E1 -11001.419,E2 -11001.419} C_VEL
LIN {X 0,Y 404.178,Z 550.127,A -85,B 0,C 180,E1 -11004.666,E2 -11004.666} C_VEL
LIN {X 0,Y 404.196,Z 550.139,A -85,B 0,C 180,E1 -11008,E2 -11008} C_VEL
LIN {X 0,Y 404.14,Z 550.135,A -85,B 0,C 180,E1 -11011.558,E2 -11011.558} C_VEL
LIN {X 0,Y 404.186,Z 550.131,A -85,B 0,C 180,E1 -11015.016,E2 -11015.016} C_VEL
LIN {X 0,Y 404.156,Z 550.139,A -85,B 0,C 180,E1 -11018.757,E2 -11018.757} C_VEL
LIN {X 0,Y 404.125,Z 550.146,A -85,B 0,C 180,E1 -11021.6,E2 -11021.6} C_VEL
LIN {X 0,Y 404.147,Z 550.144,A -85,B 0,C 180,E1 -11024.522,E2 -11024.522} C_VEL
LIN {X 0,Y 404.134,Z 550.126,A -85,B 0,C 180,E1 -11027.295,E2 -11027.295} C_VEL
LIN {X 0,Y 404.172,Z 550.142,A -85,B 0,C 180,E1 -11029.955,E2 -11029.955} C_VEL
LIN {X 0,Y 404.14,Z 550.143,A -85,B 0,C 180,E1 -11033.125,E2 -11033.125} C_VEL
LIN {X 0,Y 404.148,Z 550.145,A -85,B 0,C 180,E1 -11036.188,E2 -11036.188} C_VEL
LIN {X 0,Y 404.175,Z 550.263,A -85,B 0,C 180,E1 -11038.666,E2 -11038.666} C_VEL
LIN {X 0,Y 408.008,Z 565.832,A -85,B 0,C 180,E1 -11041.46,E2 -11041.46} C_VEL
LIN {X 0,Y 409.61,Z 573.695,A -85,B 0,C 180,E1 -11042.853,E2 -11042.853} C_VEL
LIN {X 0,Y 409.238,Z 582.764,A -85,B 0,C 180,E1 -11044.302,E2 -11044.302} C_VEL
LIN {X 0,Y 408.076,Z 603.099,A -85,B 0,C 180,E1 -11047.468,E2 -11047.468} C_VEL
LIN {X 0,Y 407.327,Z 621.909,A -85,B 0,C 180,E1 -11050.247,E2 -11050.247} C_VEL
LIN {X 0,Y 407.298,Z 622.803,A -85,B 0,C 180,E1 -11050.372,E2 -11050.372} C_VEL
LIN {X 0,Y 410.476,Z 642.724,A -85,B 0,C 180,E1 -11050.898,E2 -11050.898} C_VEL
LIN {X 0,Y 409.63,Z 718.488,A -85,B 0,C 180,E1 -11052.237,E2 -11052.237} C_VEL
LIN {X 0,Y 409.382,Z 735.767,A -85,B 0,C 180,E1 -11052.581,E2 -11052.581} C_VEL
LIN {X 0,Y 408.891,Z 748.928,A -85,B 0,C 180,E1 -11053.042,E2 -11053.042} C_VEL
LIN {X 0,Y 408.192,Z 761.538,A -85,B 0,C 180,E1 -11053.688,E2 -11053.688} C_VEL
LIN {X 0,Y 407.489,Z 773.15,A -85,B 0,C 180,E1 -11054.494,E2 -11054.494} C_VEL
LIN {X 0,Y 406.769,Z 784.883,A -85,B 0,C 180,E1 -11055.554,E2 -11055.554} C_VEL
LIN {X 0,Y 405.987,Z 795.345,A -85,B 0,C 180,E1 -11056.739,E2 -11056.739} C_VEL
LIN {X 0,Y 405.138,Z 804.219,A -85,B 0,C 180,E1 -11057.984,E2 -11057.984} C_VEL
LIN {X 0,Y 404.472,Z 812.861,A -85,B 0,C 180,E1 -11059.487,E2 -11059.487} C_VEL
LIN {X 0,Y 403.893,Z 819.813,A -85,B 0,C 180,E1 -11060.989,E2 -11060.989} C_VEL
LIN {X 0,Y 403.473,Z 825.34,A -85,B 0,C 180,E1 -11062.493,E2 -11062.493} C_VEL
LIN {X 0,Y 403.346,Z 828.065,A -85,B 0,C 180,E1 -11063.4,E2 -11063.4} C_VEL
LIN {X 0,Y 402.554,Z 830.174,A -85,B 0,C 180,E1 -11064.181,E2 -11064.181} C_VEL
LIN {X 0,Y 399.505,Z 833.047,A -85,B 0,C 180,E1 -11065.465,E2 -11065.465} C_VEL
LIN {X 0,Y 396.988,Z 834.825,A -85,B 0,C 180,E1 -11066.522,E2 -11066.522} C_VEL
LIN {X 0,Y 395.917,Z 835.86,A -85,B 0,C 180,E1 -11067.351,E2 -11067.351} C_VEL
LIN {X 0,Y 395.834,Z 836.097,A -85,B 0,C 180,E1 -11067.633,E2 -11067.633} C_VEL
LIN {X 0,Y 395.796,Z 837.037,A -85,B 0,C 180,E1 -11068.982,E2 -11068.982} C_VEL
LIN {X 0,Y 395.779,Z 837.273,A -85,B 0,C 180,E1 -11069.999,E2 -11069.999} C_VEL
LIN {X 0,Y 395.796,Z 837.082,A -85,B 0,C 180,E1 -11071.017,E2 -11071.017} C_VEL
LIN {X 0,Y 395.841,Z 836.497,A -85,B 0,C 180,E1 -11072.034,E2 -11072.034} C_VEL
LIN {X 0,Y 395.845,Z 835.532,A -85,B 0,C 180,E1 -11073.052,E2 -11073.052} C_VEL
LIN {X 0,Y 395.877,Z 834.17,A -85,B 0,C 180,E1 -11074.071,E2 -11074.071} C_VEL
LIN {X 0,Y 396.115,Z 831.299,A -85,B 0,C 180,E1 -11075.599,E2 -11075.599} C_VEL
LIN {X 0,Y 396.307,Z 827.401,A -85,B 0,C 180,E1 -11077.13,E2 -11077.13} C_VEL
LIN {X 0,Y 396.662,Z 822.354,A -85,B 0,C 180,E1 -11078.661,E2 -11078.661} C_VEL
LIN {X 0,Y 397.214,Z 815.988,A -85,B 0,C 180,E1 -11080.19,E2 -11080.19} C_VEL
LIN {X 0,Y 397.905,Z 808.068,A -85,B 0,C 180,E1 -11081.718,E2 -11081.718} C_VEL
LIN {X 0,Y 398.668,Z 799.97,A -85,B 0,C 180,E1 -11082.988,E2 -11082.988} C_VEL
LIN {X 0,Y 399.534,Z 790.032,A -85,B 0,C 180,E1 -11084.256,E2 -11084.256} C_VEL
LIN {X 0,Y 400.313,Z 778.868,A -85,B 0,C 180,E1 -11085.398,E2 -11085.398} C_VEL
LIN {X 0,Y 401.096,Z 767.924,A -85,B 0,C 180,E1 -11086.28,E2 -11086.28} C_VEL
LIN {X 0,Y 401.802,Z 755.611,A -85,B 0,C 180,E1 -11087.035,E2 -11087.035} C_VEL
LIN {X 0,Y 402.374,Z 742.808,A -85,B 0,C 180,E1 -11087.6,E2 -11087.6} C_VEL
LIN {X 0,Y 402.693,Z 730.706,A -85,B 0,C 180,E1 -11087.946,E2 -11087.946} C_VEL
LIN {X 0,Y 403.843,Z 646.312,A -85,B 0,C 180,E1 -11089.46,E2 -11089.46} C_VEL
LIN {X 0,Y 400.07,Z 623.764,A -85,B 0,C 180,E1 -11090.081,E2 -11090.081} C_VEL
LIN {X 0,Y 400.786,Z 604.74,A -85,B 0,C 180,E1 -11093.237,E2 -11093.237} C_VEL
LIN {X 0,Y 401.761,Z 588.055,A -85,B 0,C 180,E1 -11096.183,E2 -11096.183} C_VEL
LIN {X 0,Y 402.43,Z 575.849,A -85,B 0,C 180,E1 -11098.373,E2 -11098.373} C_VEL
LIN {X 0,Y 401.418,Z 569.422,A -85,B 0,C 180,E1 -11099.642,E2 -11099.642} C_VEL
LIN {X 0,Y 398.293,Z 555.736,A -85,B 0,C 180,E1 -11102.389,E2 -11102.389} C_VEL
LIN {X 0,Y 397.127,Z 551.015,A -85,B 0,C 180,E1 -11103.381,E2 -11103.381} C_VEL
LIN {X 0,Y 397.099,Z 551.022,A -85,B 0,C 180,E1 -11106.993,E2 -11106.993} C_VEL
LIN {X 0,Y 397.11,Z 551.013,A -85,B 0,C 180,E1 -11109.576,E2 -11109.576} C_VEL
LIN {X 0,Y 397.1,Z 551.007,A -85,B 0,C 180,E1 -11113.478,E2 -11113.478} C_VEL
LIN {X 0,Y 397.154,Z 551.012,A -85,B 0,C 180,E1 -11116.511,E2 -11116.511} C_VEL
LIN {X 0,Y 397.132,Z 551.018,A -85,B 0,C 180,E1 -11118.993,E2 -11118.993} C_VEL
LIN {X 0,Y 402.661,Z 566.859,A -85,B 0,C 180,E1 -11119.57,E2 -11119.57} C_VEL
LIN {X 0,Y 401.793,Z 630.943,A -85,B 0,C 180,E1 -11120.877,E2 -11120.877} C_VEL
LIN {X 0,Y 401.699,Z 644.255,A -85,B 0,C 180,E1 -11121.343,E2 -11121.343} C_VEL
LIN {X 0,Y 401.445,Z 656.815,A -85,B 0,C 180,E1 -11121.978,E2 -11121.978} C_VEL
LIN {X 0,Y 400.987,Z 668.867,A -85,B 0,C 180,E1 -11122.794,E2 -11122.794} C_VEL
LIN {X 0,Y 400.452,Z 680.708,A -85,B 0,C 180,E1 -11123.831,E2 -11123.831} C_VEL
LIN {X 0,Y 399.866,Z 691.484,A -85,B 0,C 180,E1 -11125.011,E2 -11125.011} C_VEL
LIN {X 0,Y 399.241,Z 701.093,A -85,B 0,C 180,E1 -11126.323,E2 -11126.323} C_VEL
LIN {X 0,Y 398.722,Z 709.782,A -85,B 0,C 180,E1 -11127.783,E2 -11127.783} C_VEL
LIN {X 0,Y 398.229,Z 716.718,A -85,B 0,C 180,E1 -11129.216,E2 -11129.216} C_VEL
LIN {X 0,Y 397.75,Z 723.262,A -85,B 0,C 180,E1 -11130.928,E2 -11130.928} C_VEL
LIN {X 0,Y 397.508,Z 728.256,A -85,B 0,C 180,E1 -11132.633,E2 -11132.633} C_VEL
LIN {X 0,Y 397.284,Z 732.099,A -85,B 0,C 180,E1 -11134.444,E2 -11134.444} C_VEL
LIN {X 0,Y 397.148,Z 734.261,A -85,B 0,C 180,E1 -11135.983,E2 -11135.983} C_VEL
LIN {X 0,Y 397.167,Z 735.185,A -85,B 0,C 180,E1 -11137.089,E2 -11137.089} C_VEL
LIN {X 0,Y 397.186,Z 735.671,A -85,B 0,C 180,E1 -11138.187,E2 -11138.187} C_VEL
LIN {X 0,Y 397.296,Z 735.537,A -85,B 0,C 180,E1 -11139.639,E2 -11139.639} C_VEL
LIN {X 0,Y 397.541,Z 734.226,A -85,B 0,C 180,E1 -11141.445,E2 -11141.445} C_VEL
LIN {X 0,Y 397.743,Z 732.682,A -85,B 0,C 180,E1 -11142.58,E2 -11142.58} C_VEL
LIN {X 0,Y 398.081,Z 729.733,A -85,B 0,C 180,E1 -11144.118,E2 -11144.118} C_VEL
LIN {X 0,Y 398.619,Z 725.092,A -85,B 0,C 180,E1 -11145.852,E2 -11145.852} C_VEL
LIN {X 0,Y 399.284,Z 719.031,A -85,B 0,C 180,E1 -11147.548,E2 -11147.548} C_VEL
LIN {X 0,Y 399.974,Z 711.956,A -85,B 0,C 180,E1 -11149.087,E2 -11149.087} C_VEL
LIN {X 0,Y 400.667,Z 704.445,A -85,B 0,C 180,E1 -11150.408,E2 -11150.408} C_VEL
LIN {X 0,Y 401.427,Z 695.476,A -85,B 0,C 180,E1 -11151.695,E2 -11151.695} C_VEL
LIN {X 0,Y 402.108,Z 685.547,A -85,B 0,C 180,E1 -11152.846,E2 -11152.846} C_VEL
LIN {X 0,Y 402.838,Z 673.683,A -85,B 0,C 180,E1 -11153.935,E2 -11153.935} C_VEL
LIN {X 0,Y 403.342,Z 662.529,A -85,B 0,C 180,E1 -11154.734,E2 -11154.734} C_VEL
LIN {X 0,Y 403.679,Z 649.22,A -85,B 0,C 180,E1 -11155.444,E2 -11155.444} C_VEL
LIN {X 0,Y 403.745,Z 636.689,A -85,B 0,C 180,E1 -11155.914,E2 -11155.914} C_VEL
LIN {X 0,Y 404.244,Z 600.821,A -85,B 0,C 180,E1 -11156.707,E2 -11156.707} C_VEL
LIN {X 0,Y 404.984,Z 569.352,A -85,B 0,C 180,E1 -11157.389,E2 -11157.389} C_VEL
LIN {X 0,Y 398.618,Z 554.136,A -85,B 0,C 180,E1 -11158.183,E2 -11158.183} C_VEL
LIN {X 0,Y 397.539,Z 551.676,A -85,B 0,C 180,E1 -11158.322,E2 -11158.322} C_VEL
LIN {X 0,Y 397.418,Z 550.984,A -85,B 0,C 180,E1 -11158.353,E2 -11158.353} C_VEL
LIN {X 0,Y 397.572,Z 550.964,A -85,B 0,C 180,E1 -11160,E2 -11160} C_VEL
LIN {X 0,Y 397.374,Z 550.987,A -85,B 0,C 180,E1 -11163.041,E2 -11163.041} C_VEL
LIN {X 0,Y 397.378,Z 550.985,A -85,B 0,C 180,E1 -11166.091,E2 -11166.091} C_VEL
LIN {X 0,Y 397.367,Z 550.984,A -85,B 0,C 180,E1 -11168.134,E2 -11168.134} C_VEL
LIN {X 0,Y 397.219,Z 551.005,A -85,B 0,C 180,E1 -11172.258,E2 -11172.258} C_VEL
LIN {X 0,Y 397.17,Z 551.005,A -85,B 0,C 180,E1 -11175.392,E2 -11175.392} C_VEL
LIN {X 0,Y 397.152,Z 551.015,A -85,B 0,C 180,E1 -11178.574,E2 -11178.574} C_VEL
LIN {X 0,Y 397.087,Z 551.02,A -85,B 0,C 180,E1 -11181.819,E2 -11181.819} C_VEL
LIN {X 0,Y 397.147,Z 551.015,A -85,B 0,C 180,E1 -11185.132,E2 -11185.132} C_VEL
LIN {X 0,Y 397.154,Z 551.01,A -85,B 0,C 180,E1 -11187.777,E2 -11187.777} C_VEL
LIN {X 0,Y 397.076,Z 551.025,A -85,B 0,C 180,E1 -11190.883,E2 -11190.883} C_VEL
LIN {X 0,Y 397.118,Z 551.015,A -85,B 0,C 180,E1 -11194.494,E2 -11194.494} C_VEL
LIN {X 0,Y 397.103,Z 551.017,A -85,B 0,C 180,E1 -11198.275,E2 -11198.275} C_VEL
LIN {X 0,Y 397.15,Z 551.015,A -85,B 0,C 180,E1 -11201.994,E2 -11201.994} C_VEL
LIN {X 0,Y 397.145,Z 551.015,A -85,B 0,C 180,E1 -11205.061,E2 -11205.061} C_VEL
LIN {X 0,Y 397.151,Z 551.015,A -85,B 0,C 180,E1 -11208.008,E2 -11208.008} C_VEL
LIN {X 0,Y 397.106,Z 551.021,A -85,B 0,C 180,E1 -11211.727,E2 -11211.727} C_VEL
LIN {X 0,Y 397.128,Z 551.021,A -85,B 0,C 180,E1 -11215.509,E2 -11215.509} C_VEL
LIN {X 0,Y 397.149,Z 551.256,A -85,B 0,C 180,E1 -11215.832,E2 -11215.832} C_VEL
LIN {X 0,Y 400.338,Z 563.544,A -85,B 0,C 180,E1 -11218.494,E2 -11218.494} C_VEL
LIN {X 0,Y 402.779,Z 574.966,A -85,B 0,C 180,E1 -11220.755,E2 -11220.755} C_VEL
LIN {X 0,Y 402.768,Z 578.162,A -85,B 0,C 180,E1 -11221.326,E2 -11221.326} C_VEL
LIN {X 0,Y 400.839,Z 599.27,A -85,B 0,C 180,E1 -11224.839,E2 -11224.839} C_VEL
LIN {X 0,Y 399.205,Z 622.008,A -85,B 0,C 180,E1 -11228.515,E2 -11228.515} C_VEL
LIN {X 0,Y 398.905,Z 627.148,A -85,B 0,C 180,E1 -11229.339,E2 -11229.339} C_VEL
LIN {X 0,Y 401.749,Z 650.104,A -85,B 0,C 180,E1 -11230.047,E2 -11230.047} C_VEL
LIN {X 0,Y 403.635,Z 672.458,A -85,B 0,C 180,E1 -11230.649,E2 -11230.649} C_VEL
LIN {X 0,Y 402.176,Z 741.157,A -85,B 0,C 180,E1 -11232.096,E2 -11232.096} C_VEL
LIN {X 0,Y 401.854,Z 759.207,A -85,B 0,C 180,E1 -11232.475,E2 -11232.475} C_VEL
